KUKA KRL program: PPR_fullpath_2mm_split1.src

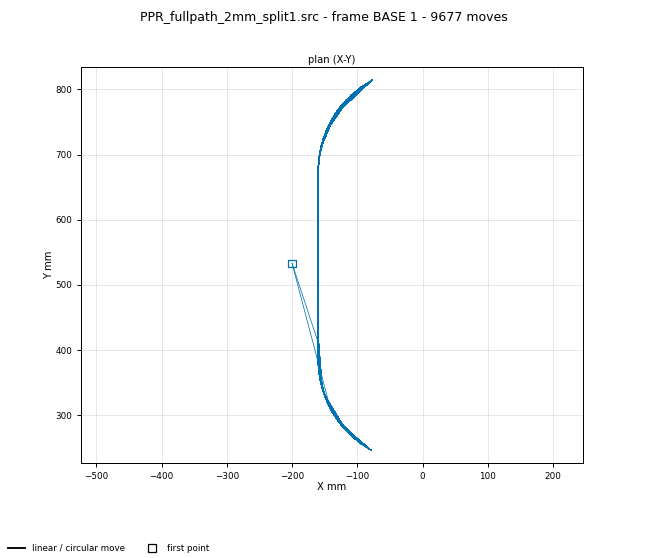
[picture p0: tool path of PPR_fullpath_2mm_split1.src in frame BASE 1, 9677 of 9678 moves have a stored position in this frame; points joined in program order, loops and branches not executed]
&ACCESS RVEO
&REL 11
&PARAM TEMPLATE = C:\KRC\Roboter\Template\vorgabe
&PARAM EDITMASK = *
DEF variable_helical2( )
;FOLD INI
  ;FOLD BASISTECH INI
    GLOBAL INTERRUPT DECL 3 WHEN $STOPMESS==TRUE DO IR_STOPM ( )
    INTERRUPT ON 3
    BAS (#INITMOV,0 )
  ;ENDFOLD (BASISTECH INI)
 ;FOLD USER INI


    ;Make your modifications here
  ;ENDFOLD (USER INI)
;ENDFOLD (INI)
ACTION(#AXIS_RESET,34,1000,#NOERROR,ERROR_CODE)
;FOLD PTP HOME  Vel= 100 % DEFAULT;%{PE}%MKUKATPBASIS,%CMOVE,%VPTP,%P 1:PTP, 2:HOME, 3:, 5:100, 7:DEFAULT
$BWDSTART = FALSE
PDAT_ACT=PDEFAULT
FDAT_ACT=FHOME
BAS (#PTP_PARAMS,100 )
$H_POS=XHOME
PTP  XHOME
;ENDFOLD
BAS(#TOOL,1)
BAS(#BASE,1)
$VEL_AXIS[1]=100
$VEL_AXIS[2]=100
$VEL_AXIS[3]=100
$VEL_AXIS[4]=100
$VEL_AXIS[5]=100
$VEL_AXIS[6]=100
$VEL_EXTAX[1]=100
$VEL_EXTAX[2]=100

$ACC_AXIS[1]=100
$ACC_AXIS[2]=100
$ACC_AXIS[3]=100
$ACC_AXIS[4]=100
$ACC_AXIS[5]=100
$ACC_AXIS[6]=100
$ACC_EXTAX[1]=100
$ACC_EXTAX[2]=100

SLIN {X  -200.000, Y  +533.000, Z    +0.000, A    +0.000, E1    +0.000, E3    +0.000, E4    +0.000}

SLIN {X  -141.408, Y  +310.842, Z    +0.000, E1   +71.243, E3  -388.598}
HALT
SPLINE
SPL {X  -134.330, Y  +298.778, Z    +0.000, E1   +70.323, E3  -374.632}
SPL {X  -128.957, Y  +290.989, Z    +0.000, E1   +69.528, E3  -365.267}
SPL {X  -124.846, Y  +285.632, Z    +0.000, E1   +68.906, E3  -358.804}
SPL {X  -121.783, Y  +281.927, Z    +0.000, E1   +68.403, E3  -354.372}
SPL {X   -79.219, Y  +246.688, Z    +0.000, E1   +55.887, E3  -232.865}
ENDSPLINE

SPLINE
SPL {X  -125.038, Y  +285.873, Z    +0.000, E1   +53.023, E3   -55.824}
SPL {X  -149.949, Y  +329.886, Z    +0.000, E1   +41.515, E3   -34.259}
SPL {X  -157.246, Y  +356.141, Z    +0.000, E1   +27.282, E3   -29.202}
SPL {X  -159.525, Y  +373.376, Z    +0.000, E1   +13.812, E3   -27.545}
SPL {X  -160.000, Y  +387.264, Z    +0.000, E1    +0.544, E3   -27.088}
SPL {X  -160.000, Y  +390.384, Z    +0.000, E1    -6.008, E3   -27.050}
SPL {X  -160.000, Y  +395.752, Z    +0.000, E1   -19.038, E3   -26.857}
SPL {X  -160.000, Y  +404.289, Z    +0.000, E1   -38.292, E3   -26.188}
SPL {X  -160.000, Y  +418.681, Z    +0.000, E1   -56.949, E3   -23.999}
SPL {X  -160.000, Y  +471.977, Z    +0.000, E1   -70.792, E3    -7.479}
SPL {X  -159.977, Y  +677.138, Z    +0.000, E1   -73.665, E3   +89.012}
SPL {X  -157.805, Y  +700.810, Z    +0.000, E1   -73.511, E3  +105.842}
SPL {X  -152.242, Y  +723.618, Z    +0.000, E1   -72.940, E3  +125.755}
SPL {X  -145.929, Y  +740.010, Z    +0.000, E1   -72.229, E3  +142.226}
SPL {X  -139.114, Y  +753.439, Z    +0.000, E1   -71.436, E3  +156.865}
SPL {X  -132.333, Y  +764.333, Z    +0.000, E1   -70.535, E3  +169.489}
SPL {X  -125.486, Y  +773.664, Z    +0.000, E1   -69.598, E3  +180.463}
SPL {X  -121.321, Y  +778.713, Z    +0.000, E1   -68.872, E3  +186.473}
SPL {X   -77.337, Y  +814.468, Z    +0.000, E1   -56.377, E3  +305.104}
ENDSPLINE

SPLINE
SPL {X  -134.727, Y  +760.706, Z    +0.000, E1   -50.460, E3  +493.336}
SPL {X  -155.580, Y  +711.748, Z    +0.000, E1   -32.084, E3  +510.251}
SPL {X  -159.445, Y  +687.715, Z    +0.000, E1   -14.660, E3  +513.097}
SPL {X  -159.995, Y  +675.725, Z    +0.000, E1    -3.424, E3  +513.608}
SPL {X  -160.000, Y  +671.714, Z    +0.000, E1    +0.835, E3  +513.649}
SPL {X  -160.000, Y  +663.084, Z    +0.000, E1   +21.134, E3  +513.973}
SPL {X  -160.000, Y  +650.910, Z    +0.000, E1   +46.005, E3  +515.127}
SPL {X  -160.000, Y  +634.843, Z    +0.000, E1   +61.273, E3  +517.804}
SPL {X  -160.000, Y  +578.679, Z    +0.000, E1   +71.665, E3  +535.637}
SPL {X  -160.000, Y  +387.528, Z    +0.000, E1   +73.487, E3  +628.450}
SPL {X  -159.218, Y  +369.903, Z    +0.000, E1   +73.425, E3  +640.317}
SPL {X  -156.808, Y  +353.900, Z    +0.000, E1   +73.180, E3  +652.921}
SPL {X  -154.539, Y  +344.254, Z    +0.000, E1   +72.827, E3  +662.458}
ENDSPLINE

SPLINE
SPL {X  -157.258, Y  +356.206, Z    +0.000, E1   +70.434, E3  +677.030}
ENDSPLINE

SPLINE
SPL {X  -150.342, Y  +330.952, Z    +0.000, E1   +71.154, E3  +688.703}
SPL {X  -141.358, Y  +310.748, Z    +0.000, E1   +71.233, E3  +701.409}
SPL {X  -134.330, Y  +298.778, Z    +0.000, E1   +70.323, E3  +715.256}
SPL {X  -128.957, Y  +290.989, Z    +0.000, E1   +69.528, E3  +724.621}
SPL {X  -124.846, Y  +285.632, Z    +0.000, E1   +68.906, E3  +731.084}
SPL {X  -121.783, Y  +281.927, Z    +0.000, E1   +68.403, E3  +735.517}
SPL {X   -79.219, Y  +246.688, Z    +0.000, E1   +55.887, E3  +857.023}
ENDSPLINE

SPLINE
SPL {X  -125.038, Y  +285.873, Z    +0.000, E1   +53.023, E3 +1034.064}
SPL {X  -149.949, Y  +329.886, Z    +0.000, E1   +41.515, E3 +1055.629}
SPL {X  -157.246, Y  +356.141, Z    +0.000, E1   +27.282, E3 +1060.686}
SPL {X  -159.525, Y  +373.376, Z    +0.000, E1   +13.812, E3 +1062.343}
SPL {X  -160.000, Y  +387.264, Z    +0.000, E1    +0.544, E3 +1062.800}
SPL {X  -160.000, Y  +390.384, Z    +0.000, E1    -6.008, E3 +1062.838}
SPL {X  -160.000, Y  +395.752, Z    +0.000, E1   -19.038, E3 +1063.031}
SPL {X  -160.000, Y  +404.289, Z    +0.000, E1   -38.292, E3 +1063.700}
SPL {X  -160.000, Y  +418.681, Z    +0.000, E1   -56.949, E3 +1065.889}
SPL {X  -160.000, Y  +471.977, Z    +0.000, E1   -70.792, E3 +1082.409}
SPL {X  -159.977, Y  +677.138, Z    +0.000, E1   -73.665, E3 +1178.900}
SPL {X  -157.805, Y  +700.810, Z    +0.000, E1   -73.511, E3 +1195.730}
SPL {X  -152.242, Y  +723.618, Z    +0.000, E1   -72.940, E3 +1215.643}
SPL {X  -145.929, Y  +740.010, Z    +0.000, E1   -72.229, E3 +1232.114}
SPL {X  -139.114, Y  +753.439, Z    +0.000, E1   -71.436, E3 +1246.753}
SPL {X  -132.333, Y  +764.333, Z    +0.000, E1   -70.535, E3 +1259.377}
SPL {X  -125.486, Y  +773.664, Z    +0.000, E1   -69.598, E3 +1270.351}
SPL {X  -121.321, Y  +778.713, Z    +0.000, E1   -68.872, E3 +1276.361}
SPL {X   -77.337, Y  +814.468, Z    +0.000, E1   -56.377, E3 +1394.992}
ENDSPLINE

SPLINE
SPL {X  -134.727, Y  +760.706, Z    +0.000, E1   -50.460, E3 +1583.224}
SPL {X  -155.580, Y  +711.748, Z    +0.000, E1   -32.084, E3 +1600.139}
SPL {X  -159.445, Y  +687.715, Z    +0.000, E1   -14.660, E3 +1602.986}
SPL {X  -159.995, Y  +675.725, Z    +0.000, E1    -3.424, E3 +1603.496}
SPL {X  -160.000, Y  +671.714, Z    +0.000, E1    +0.835, E3 +1603.537}
SPL {X  -160.000, Y  +663.084, Z    +0.000, E1   +21.134, E3 +1603.861}
SPL {X  -160.000, Y  +650.910, Z    +0.000, E1   +46.005, E3 +1605.015}
SPL {X  -160.000, Y  +634.843, Z    +0.000, E1   +61.273, E3 +1607.692}
SPL {X  -160.000, Y  +578.679, Z    +0.000, E1   +71.665, E3 +1625.525}
SPL {X  -160.000, Y  +387.528, Z    +0.000, E1   +73.487, E3 +1718.338}
SPL {X  -159.218, Y  +369.903, Z    +0.000, E1   +73.425, E3 +1730.205}
SPL {X  -156.808, Y  +353.900, Z    +0.000, E1   +73.180, E3 +1742.809}
SPL {X  -154.539, Y  +344.254, Z    +0.000, E1   +72.827, E3 +1752.346}
ENDSPLINE

SPLINE
SPL {X  -157.258, Y  +356.206, Z    +0.000, E1   +70.434, E3 +1766.919}
ENDSPLINE

SPLINE
SPL {X  -150.342, Y  +330.952, Z    +0.000, E1   +71.154, E3 +1778.591}
SPL {X  -141.358, Y  +310.748, Z    +0.000, E1   +71.233, E3 +1791.297}
SPL {X  -134.330, Y  +298.778, Z    +0.000, E1   +70.323, E3 +1805.144}
SPL {X  -128.957, Y  +290.989, Z    +0.000, E1   +69.528, E3 +1814.509}
SPL {X  -124.846, Y  +285.632, Z    +0.000, E1   +68.906, E3 +1820.972}
SPL {X  -121.783, Y  +281.927, Z    +0.000, E1   +68.403, E3 +1825.405}
SPL {X   -79.219, Y  +246.688, Z    +0.000, E1   +55.887, E3 +1946.911}
ENDSPLINE

SPLINE
SPL {X  -125.038, Y  +285.873, Z    +0.000, E1   +53.023, E3 +2123.952}
SPL {X  -149.949, Y  +329.886, Z    +0.000, E1   +41.515, E3 +2145.517}
SPL {X  -157.246, Y  +356.141, Z    +0.000, E1   +27.282, E3 +2150.574}
SPL {X  -159.525, Y  +373.376, Z    +0.000, E1   +13.812, E3 +2152.231}
SPL {X  -160.000, Y  +387.264, Z    +0.000, E1    +0.544, E3 +2152.688}
SPL {X  -160.000, Y  +390.384, Z    +0.000, E1    -6.008, E3 +2152.726}
SPL {X  -160.000, Y  +395.752, Z    +0.000, E1   -19.038, E3 +2152.919}
SPL {X  -160.000, Y  +404.289, Z    +0.000, E1   -38.292, E3 +2153.588}
SPL {X  -160.000, Y  +418.681, Z    +0.000, E1   -56.949, E3 +2155.777}
SPL {X  -160.000, Y  +471.977, Z    +0.000, E1   -70.792, E3 +2172.297}
SPL {X  -159.977, Y  +677.138, Z    +0.000, E1   -73.665, E3 +2268.788}
SPL {X  -157.805, Y  +700.810, Z    +0.000, E1   -73.511, E3 +2285.618}
SPL {X  -152.242, Y  +723.618, Z    +0.000, E1   -72.940, E3 +2305.531}
SPL {X  -145.929, Y  +740.010, Z    +0.000, E1   -72.229, E3 +2322.002}
SPL {X  -139.114, Y  +753.439, Z    +0.000, E1   -71.436, E3 +2336.641}
SPL {X  -132.333, Y  +764.333, Z    +0.000, E1   -70.535, E3 +2349.265}
SPL {X  -125.486, Y  +773.664, Z    +0.000, E1   -69.598, E3 +2360.239}
SPL {X  -121.321, Y  +778.713, Z    +0.000, E1   -68.872, E3 +2366.249}
SPL {X   -77.337, Y  +814.468, Z    +0.000, E1   -56.377, E3 +2484.880}
ENDSPLINE

SPLINE
SPL {X  -134.727, Y  +760.706, Z    +0.000, E1   -50.460, E3 +2673.112}
SPL {X  -155.580, Y  +711.748, Z    +0.000, E1   -32.084, E3 +2690.027}
SPL {X  -159.445, Y  +687.715, Z    +0.000, E1   -14.660, E3 +2692.874}
SPL {X  -159.995, Y  +675.725, Z    +0.000, E1    -3.424, E3 +2693.384}
SPL {X  -160.000, Y  +671.714, Z    +0.000, E1    +0.835, E3 +2693.425}
SPL {X  -160.000, Y  +663.084, Z    +0.000, E1   +21.134, E3 +2693.749}
SPL {X  -160.000, Y  +650.910, Z    +0.000, E1   +46.005, E3 +2694.903}
SPL {X  -160.000, Y  +634.843, Z    +0.000, E1   +61.273, E3 +2697.580}
SPL {X  -160.000, Y  +578.679, Z    +0.000, E1   +71.665, E3 +2715.413}
SPL {X  -160.000, Y  +387.528, Z    +0.000, E1   +73.487, E3 +2808.226}
SPL {X  -159.218, Y  +369.903, Z    +0.000, E1   +73.425, E3 +2820.093}
SPL {X  -156.808, Y  +353.900, Z    +0.000, E1   +73.180, E3 +2832.697}
SPL {X  -154.539, Y  +344.254, Z    +0.000, E1   +72.827, E3 +2842.234}
ENDSPLINE

SPLINE
SPL {X  -157.258, Y  +356.206, Z    +0.000, E1   +70.434, E3 +2856.807}
ENDSPLINE

SPLINE
SPL {X  -150.342, Y  +330.952, Z    +0.000, E1   +71.154, E3 +2868.479}
SPL {X  -141.358, Y  +310.748, Z    +0.000, E1   +71.233, E3 +2881.185}
SPL {X  -134.330, Y  +298.778, Z    +0.000, E1   +70.323, E3 +2895.032}
SPL {X  -128.957, Y  +290.989, Z    +0.000, E1   +69.528, E3 +2904.397}
SPL {X  -124.846, Y  +285.632, Z    +0.000, E1   +68.906, E3 +2910.860}
SPL {X  -121.783, Y  +281.927, Z    +0.000, E1   +68.403, E3 +2915.293}
SPL {X   -79.219, Y  +246.688, Z    +0.000, E1   +55.887, E3 +3036.799}
ENDSPLINE

SPLINE
SPL {X  -125.038, Y  +285.873, Z    +0.000, E1   +53.023, E3 +3213.840}
SPL {X  -149.949, Y  +329.886, Z    +0.000, E1   +41.515, E3 +3235.405}
SPL {X  -157.246, Y  +356.141, Z    +0.000, E1   +27.282, E3 +3240.462}
SPL {X  -159.525, Y  +373.376, Z    +0.000, E1   +13.812, E3 +3242.119}
SPL {X  -160.000, Y  +387.264, Z    +0.000, E1    +0.544, E3 +3242.577}
SPL {X  -160.000, Y  +390.384, Z    +0.000, E1    -6.008, E3 +3242.614}
SPL {X  -160.000, Y  +395.752, Z    +0.000, E1   -19.038, E3 +3242.807}
SPL {X  -160.000, Y  +404.289, Z    +0.000, E1   -38.292, E3 +3243.476}
SPL {X  -160.000, Y  +418.681, Z    +0.000, E1   -56.949, E3 +3245.665}
SPL {X  -160.000, Y  +458.961, Z    +0.000, E1   -69.778, E3 +3257.262}
SPL {X  -160.000, Y  +485.343, Z    +0.000, E1   -71.539, E3 +3267.248}
SPL {X  -159.977, Y  +677.138, Z    +0.000, E1   -73.665, E3 +3358.676}
SPL {X  -157.805, Y  +700.810, Z    +0.000, E1   -73.511, E3 +3375.506}
SPL {X  -152.242, Y  +723.618, Z    +0.000, E1   -72.940, E3 +3395.419}
SPL {X  -145.929, Y  +740.010, Z    +0.000, E1   -72.229, E3 +3411.890}
SPL {X  -139.114, Y  +753.439, Z    +0.000, E1   -71.436, E3 +3426.529}
SPL {X  -132.333, Y  +764.333, Z    +0.000, E1   -70.535, E3 +3439.153}
SPL {X  -125.486, Y  +773.664, Z    +0.000, E1   -69.598, E3 +3450.127}
SPL {X  -121.321, Y  +778.713, Z    +0.000, E1   -68.872, E3 +3456.137}
SPL {X   -77.337, Y  +814.468, Z    +0.000, E1   -56.377, E3 +3574.768}
ENDSPLINE

SPLINE
SPL {X  -134.727, Y  +760.706, Z    +0.000, E1   -50.460, E3 +3763.000}
SPL {X  -155.580, Y  +711.748, Z    +0.000, E1   -32.084, E3 +3779.915}
SPL {X  -159.445, Y  +687.715, Z    +0.000, E1   -14.660, E3 +3782.762}
SPL {X  -159.995, Y  +675.725, Z    +0.000, E1    -3.424, E3 +3783.272}
SPL {X  -160.000, Y  +671.714, Z    +0.000, E1    +0.835, E3 +3783.313}
SPL {X  -160.000, Y  +663.084, Z    +0.000, E1   +21.134, E3 +3783.637}
SPL {X  -160.000, Y  +650.910, Z    +0.000, E1   +46.005, E3 +3784.791}
SPL {X  -160.000, Y  +634.843, Z    +0.000, E1   +61.273, E3 +3787.468}
SPL {X  -160.000, Y  +578.679, Z    +0.000, E1   +71.665, E3 +3805.301}
SPL {X  -160.000, Y  +387.528, Z    +0.000, E1   +73.487, E3 +3898.114}
SPL {X  -159.218, Y  +369.903, Z    +0.000, E1   +73.425, E3 +3909.981}
SPL {X  -156.808, Y  +353.900, Z    +0.000, E1   +73.180, E3 +3922.585}
SPL {X  -154.539, Y  +344.254, Z    +0.000, E1   +72.827, E3 +3932.122}
ENDSPLINE

SPLINE
SPL {X  -157.258, Y  +356.206, Z    +0.000, E1   +70.434, E3 +3946.695}
ENDSPLINE

SPLINE
SPL {X  -150.342, Y  +330.952, Z    +0.000, E1   +71.154, E3 +3958.367}
SPL {X  -141.358, Y  +310.748, Z    +0.000, E1   +71.233, E3 +3971.073}
SPL {X  -134.330, Y  +298.778, Z    +0.000, E1   +70.323, E3 +3984.920}
SPL {X  -128.957, Y  +290.989, Z    +0.000, E1   +69.528, E3 +3994.285}
SPL {X  -124.846, Y  +285.632, Z    +0.000, E1   +68.906, E3 +4000.748}
SPL {X  -121.783, Y  +281.927, Z    +0.000, E1   +68.403, E3 +4005.181}
SPL {X   -79.219, Y  +246.688, Z    +0.000, E1   +55.887, E3 +4126.687}
ENDSPLINE

SPLINE
SPL {X  -125.038, Y  +285.873, Z    +0.000, E1   +53.023, E3 +4303.728}
SPL {X  -149.949, Y  +329.886, Z    +0.000, E1   +41.515, E3 +4325.293}
SPL {X  -157.246, Y  +356.141, Z    +0.000, E1   +27.282, E3 +4330.350}
SPL {X  -159.525, Y  +373.376, Z    +0.000, E1   +13.812, E3 +4332.007}
SPL {X  -160.000, Y  +387.264, Z    +0.000, E1    +0.544, E3 +4332.465}
SPL {X  -160.000, Y  +390.384, Z    +0.000, E1    -6.008, E3 +4332.502}
SPL {X  -160.000, Y  +395.752, Z    +0.000, E1   -19.038, E3 +4332.695}
SPL {X  -160.000, Y  +404.289, Z    +0.000, E1   -38.292, E3 +4333.364}
SPL {X  -160.000, Y  +418.681, Z    +0.000, E1   -56.949, E3 +4335.554}
SPL {X  -160.000, Y  +471.977, Z    +0.000, E1   -70.792, E3 +4352.073}
SPL {X  -159.977, Y  +677.138, Z    +0.000, E1   -73.665, E3 +4448.564}
SPL {X  -157.805, Y  +700.810, Z    +0.000, E1   -73.511, E3 +4465.394}
SPL {X  -152.242, Y  +723.618, Z    +0.000, E1   -72.940, E3 +4485.307}
SPL {X  -145.929, Y  +740.010, Z    +0.000, E1   -72.229, E3 +4501.778}
SPL {X  -139.114, Y  +753.439, Z    +0.000, E1   -71.436, E3 +4516.417}
SPL {X  -132.333, Y  +764.333, Z    +0.000, E1   -70.535, E3 +4529.041}
SPL {X  -125.486, Y  +773.664, Z    +0.000, E1   -69.598, E3 +4540.015}
SPL {X  -121.321, Y  +778.713, Z    +0.000, E1   -68.872, E3 +4546.025}
SPL {X   -77.337, Y  +814.468, Z    +0.000, E1   -56.377, E3 +4664.656}
ENDSPLINE

SPLINE
SPL {X  -134.727, Y  +760.706, Z    +0.000, E1   -50.460, E3 +4852.888}
SPL {X  -155.580, Y  +711.748, Z    +0.000, E1   -32.084, E3 +4869.803}
SPL {X  -159.445, Y  +687.715, Z    +0.000, E1   -14.660, E3 +4872.650}
SPL {X  -159.995, Y  +675.725, Z    +0.000, E1    -3.424, E3 +4873.160}
SPL {X  -160.000, Y  +671.714, Z    +0.000, E1    +0.835, E3 +4873.201}
SPL {X  -160.000, Y  +663.084, Z    +0.000, E1   +21.134, E3 +4873.525}
SPL {X  -160.000, Y  +650.910, Z    +0.000, E1   +46.005, E3 +4874.679}
SPL {X  -160.000, Y  +634.843, Z    +0.000, E1   +61.273, E3 +4877.356}
SPL {X  -160.000, Y  +578.679, Z    +0.000, E1   +71.665, E3 +4895.189}
SPL {X  -160.000, Y  +387.528, Z    +0.000, E1   +73.487, E3 +4988.002}
SPL {X  -159.218, Y  +369.903, Z    +0.000, E1   +73.425, E3 +4999.869}
SPL {X  -156.808, Y  +353.900, Z    +0.000, E1   +73.180, E3 +5012.473}
SPL {X  -154.539, Y  +344.254, Z    +0.000, E1   +72.827, E3 +5022.010}
ENDSPLINE

SPLINE
SPL {X  -157.258, Y  +356.206, Z    +0.000, E1   +70.434, E3 +5036.583}
ENDSPLINE

SPLINE
SPL {X  -150.342, Y  +330.952, Z    +0.000, E1   +71.154, E3 +5048.255}
SPL {X  -141.358, Y  +310.748, Z    +0.000, E1   +71.233, E3 +5060.961}
SPL {X  -134.330, Y  +298.778, Z    +0.000, E1   +70.323, E3 +5074.808}
SPL {X  -128.957, Y  +290.989, Z    +0.000, E1   +69.528, E3 +5084.173}
SPL {X  -124.846, Y  +285.632, Z    +0.000, E1   +68.906, E3 +5090.636}
SPL {X  -121.783, Y  +281.927, Z    +0.000, E1   +68.403, E3 +5095.069}
SPL {X   -79.219, Y  +246.688, Z    +0.000, E1   +55.887, E3 +5216.575}
ENDSPLINE

SPLINE
SPL {X  -125.038, Y  +285.873, Z    +0.000, E1   +53.023, E3 +5393.616}
SPL {X  -149.949, Y  +329.886, Z    +0.000, E1   +41.515, E3 +5415.181}
SPL {X  -157.246, Y  +356.141, Z    +0.000, E1   +27.282, E3 +5420.238}
SPL {X  -159.525, Y  +373.376, Z    +0.000, E1   +13.812, E3 +5421.895}
SPL {X  -160.000, Y  +387.264, Z    +0.000, E1    +0.544, E3 +5422.353}
SPL {X  -160.000, Y  +390.384, Z    +0.000, E1    -6.008, E3 +5422.390}
SPL {X  -160.000, Y  +395.752, Z    +0.000, E1   -19.038, E3 +5422.583}
SPL {X  -160.000, Y  +404.289, Z    +0.000, E1   -38.292, E3 +5423.252}
SPL {X  -160.000, Y  +418.681, Z    +0.000, E1   -56.949, E3 +5425.442}
SPL {X  -160.000, Y  +471.977, Z    +0.000, E1   -70.792, E3 +5441.961}
SPL {X  -159.977, Y  +677.138, Z    +0.000, E1   -73.665, E3 +5538.452}
SPL {X  -157.805, Y  +700.810, Z    +0.000, E1   -73.511, E3 +5555.282}
SPL {X  -152.242, Y  +723.618, Z    +0.000, E1   -72.940, E3 +5575.195}
SPL {X  -145.929, Y  +740.010, Z    +0.000, E1   -72.229, E3 +5591.666}
SPL {X  -139.114, Y  +753.439, Z    +0.000, E1   -71.436, E3 +5606.305}
SPL {X  -132.333, Y  +764.333, Z    +0.000, E1   -70.535, E3 +5618.929}
SPL {X  -125.486, Y  +773.664, Z    +0.000, E1   -69.598, E3 +5629.903}
SPL {X  -121.321, Y  +778.713, Z    +0.000, E1   -68.872, E3 +5635.913}
SPL {X   -77.337, Y  +814.468, Z    +0.000, E1   -56.377, E3 +5754.544}
ENDSPLINE

SPLINE
SPL {X  -134.727, Y  +760.706, Z    +0.000, E1   -50.460, E3 +5942.776}
SPL {X  -155.580, Y  +711.748, Z    +0.000, E1   -32.084, E3 +5959.691}
SPL {X  -159.445, Y  +687.715, Z    +0.000, E1   -14.660, E3 +5962.538}
SPL {X  -159.995, Y  +675.725, Z    +0.000, E1    -3.424, E3 +5963.048}
SPL {X  -160.000, Y  +671.714, Z    +0.000, E1    +0.835, E3 +5963.089}
SPL {X  -160.000, Y  +663.084, Z    +0.000, E1   +21.134, E3 +5963.413}
SPL {X  -160.000, Y  +650.910, Z    +0.000, E1   +46.005, E3 +5964.567}
SPL {X  -160.000, Y  +634.843, Z    +0.000, E1   +61.273, E3 +5967.244}
SPL {X  -160.000, Y  +578.679, Z    +0.000, E1   +71.665, E3 +5985.078}
SPL {X  -160.000, Y  +387.528, Z    +0.000, E1   +73.487, E3 +6077.890}
SPL {X  -159.218, Y  +369.903, Z    +0.000, E1   +73.425, E3 +6089.757}
SPL {X  -156.808, Y  +353.900, Z    +0.000, E1   +73.180, E3 +6102.361}
SPL {X  -154.539, Y  +344.254, Z    +0.000, E1   +72.827, E3 +6111.898}
ENDSPLINE

SPLINE
SPL {X  -157.258, Y  +356.206, Z    +0.000, E1   +70.434, E3 +6126.471}
ENDSPLINE

SPLINE
SPL {X  -150.342, Y  +330.952, Z    +0.000, E1   +71.154, E3 +6138.143}
SPL {X  -141.358, Y  +310.748, Z    +0.000, E1   +71.233, E3 +6150.849}
SPL {X  -134.330, Y  +298.778, Z    +0.000, E1   +70.323, E3 +6164.696}
SPL {X  -128.957, Y  +290.989, Z    +0.000, E1   +69.528, E3 +6174.061}
SPL {X  -124.846, Y  +285.632, Z    +0.000, E1   +68.906, E3 +6180.524}
SPL {X  -121.783, Y  +281.927, Z    +0.000, E1   +68.403, E3 +6184.957}
SPL {X   -79.219, Y  +246.688, Z    +0.000, E1   +55.887, E3 +6306.463}
ENDSPLINE

SPLINE
SPL {X  -125.038, Y  +285.873, Z    +0.000, E1   +53.023, E3 +6483.504}
SPL {X  -149.949, Y  +329.886, Z    +0.000, E1   +41.515, E3 +6505.069}
SPL {X  -157.246, Y  +356.141, Z    +0.000, E1   +27.282, E3 +6510.126}
SPL {X  -159.525, Y  +373.376, Z    +0.000, E1   +13.812, E3 +6511.783}
SPL {X  -160.000, Y  +387.264, Z    +0.000, E1    +0.544, E3 +6512.241}
SPL {X  -160.000, Y  +390.384, Z    +0.000, E1    -6.008, E3 +6512.278}
SPL {X  -160.000, Y  +395.752, Z    +0.000, E1   -19.038, E3 +6512.471}
SPL {X  -160.000, Y  +404.289, Z    +0.000, E1   -38.292, E3 +6513.140}
SPL {X  -160.000, Y  +418.681, Z    +0.000, E1   -56.949, E3 +6515.330}
SPL {X  -160.000, Y  +458.961, Z    +0.000, E1   -69.778, E3 +6526.926}
SPL {X  -160.000, Y  +485.343, Z    +0.000, E1   -71.539, E3 +6536.912}
SPL {X  -159.977, Y  +677.138, Z    +0.000, E1   -73.665, E3 +6628.340}
SPL {X  -157.805, Y  +700.810, Z    +0.000, E1   -73.511, E3 +6645.170}
SPL {X  -152.242, Y  +723.618, Z    +0.000, E1   -72.940, E3 +6665.083}
SPL {X  -145.929, Y  +740.010, Z    +0.000, E1   -72.229, E3 +6681.554}
SPL {X  -139.114, Y  +753.439, Z    +0.000, E1   -71.436, E3 +6696.193}
SPL {X  -132.333, Y  +764.333, Z    +0.000, E1   -70.535, E3 +6708.817}
SPL {X  -125.486, Y  +773.664, Z    +0.000, E1   -69.598, E3 +6719.791}
SPL {X  -121.321, Y  +778.713, Z    +0.000, E1   -68.872, E3 +6725.801}
SPL {X   -77.337, Y  +814.468, Z    +0.000, E1   -56.377, E3 +6844.432}
ENDSPLINE

SPLINE
SPL {X  -134.727, Y  +760.706, Z    +0.000, E1   -50.460, E3 +7032.664}
SPL {X  -155.580, Y  +711.748, Z    +0.000, E1   -32.084, E3 +7049.579}
SPL {X  -159.445, Y  +687.715, Z    +0.000, E1   -14.660, E3 +7052.426}
SPL {X  -159.995, Y  +675.725, Z    +0.000, E1    -3.424, E3 +7052.937}
SPL {X  -160.000, Y  +671.714, Z    +0.000, E1    +0.835, E3 +7052.977}
SPL {X  -160.000, Y  +663.084, Z    +0.000, E1   +21.134, E3 +7053.301}
SPL {X  -160.000, Y  +650.910, Z    +0.000, E1   +46.005, E3 +7054.455}
SPL {X  -160.000, Y  +634.843, Z    +0.000, E1   +61.273, E3 +7057.132}
SPL {X  -160.000, Y  +578.679, Z    +0.000, E1   +71.665, E3 +7074.966}
SPL {X  -160.000, Y  +387.528, Z    +0.000, E1   +73.487, E3 +7167.778}
SPL {X  -159.218, Y  +369.903, Z    +0.000, E1   +73.425, E3 +7179.645}
SPL {X  -156.808, Y  +353.900, Z    +0.000, E1   +73.180, E3 +7192.249}
SPL {X  -154.539, Y  +344.254, Z    +0.000, E1   +72.827, E3 +7201.786}
ENDSPLINE

SPLINE
SPL {X  -157.258, Y  +356.206, Z    +0.000, E1   +70.434, E3 +7216.359}
ENDSPLINE

SPLINE
SPL {X  -150.342, Y  +330.952, Z    +0.000, E1   +71.154, E3 +7228.031}
SPL {X  -141.358, Y  +310.748, Z    +0.000, E1   +71.233, E3 +7240.737}
SPL {X  -134.330, Y  +298.778, Z    +0.000, E1   +70.323, E3 +7254.584}
SPL {X  -128.957, Y  +290.989, Z    +0.000, E1   +69.528, E3 +7263.949}
SPL {X  -124.846, Y  +285.632, Z    +0.000, E1   +68.906, E3 +7270.413}
SPL {X  -121.783, Y  +281.927, Z    +0.000, E1   +68.403, E3 +7274.845}
SPL {X   -79.219, Y  +246.688, Z    +0.000, E1   +55.887, E3 +7396.351}
ENDSPLINE

SPLINE
SPL {X  -125.038, Y  +285.873, Z    +0.000, E1   +53.023, E3 +7573.392}
SPL {X  -149.949, Y  +329.886, Z    +0.000, E1   +41.515, E3 +7594.957}
SPL {X  -157.246, Y  +356.141, Z    +0.000, E1   +27.282, E3 +7600.014}
SPL {X  -159.525, Y  +373.376, Z    +0.000, E1   +13.812, E3 +7601.671}
SPL {X  -160.000, Y  +387.264, Z    +0.000, E1    +0.544, E3 +7602.129}
SPL {X  -160.000, Y  +390.384, Z    +0.000, E1    -6.008, E3 +7602.166}
SPL {X  -160.000, Y  +395.752, Z    +0.000, E1   -19.038, E3 +7602.359}
SPL {X  -160.000, Y  +404.289, Z    +0.000, E1   -38.292, E3 +7603.028}
SPL {X  -160.000, Y  +418.681, Z    +0.000, E1   -56.949, E3 +7605.218}
SPL {X  -160.000, Y  +471.977, Z    +0.000, E1   -70.792, E3 +7621.737}
SPL {X  -159.977, Y  +677.138, Z    +0.000, E1   -73.665, E3 +7718.228}
SPL {X  -157.805, Y  +700.810, Z    +0.000, E1   -73.511, E3 +7735.058}
SPL {X  -152.242, Y  +723.618, Z    +0.000, E1   -72.940, E3 +7754.971}
SPL {X  -145.929, Y  +740.010, Z    +0.000, E1   -72.229, E3 +7771.442}
SPL {X  -139.114, Y  +753.439, Z    +0.000, E1   -71.436, E3 +7786.081}
SPL {X  -132.333, Y  +764.333, Z    +0.000, E1   -70.535, E3 +7798.705}
SPL {X  -125.486, Y  +773.664, Z    +0.000, E1   -69.598, E3 +7809.679}
SPL {X  -121.321, Y  +778.713, Z    +0.000, E1   -68.872, E3 +7815.689}
SPL {X   -77.337, Y  +814.468, Z    +0.000, E1   -56.377, E3 +7934.320}
ENDSPLINE

SPLINE
SPL {X  -134.727, Y  +760.706, Z    +0.000, E1   -50.460, E3 +8122.552}
SPL {X  -155.580, Y  +711.748, Z    +0.000, E1   -32.084, E3 +8139.467}
SPL {X  -159.445, Y  +687.715, Z    +0.000, E1   -14.660, E3 +8142.314}
SPL {X  -159.995, Y  +675.725, Z    +0.000, E1    -3.424, E3 +8142.825}
SPL {X  -160.000, Y  +671.714, Z    +0.000, E1    +0.835, E3 +8142.865}
SPL {X  -160.000, Y  +663.084, Z    +0.000, E1   +21.134, E3 +8143.189}
SPL {X  -160.000, Y  +650.910, Z    +0.000, E1   +46.005, E3 +8144.343}
SPL {X  -160.000, Y  +634.843, Z    +0.000, E1   +61.273, E3 +8147.020}
SPL {X  -160.000, Y  +578.679, Z    +0.000, E1   +71.665, E3 +8164.854}
SPL {X  -160.000, Y  +387.528, Z    +0.000, E1   +73.487, E3 +8257.666}
SPL {X  -159.218, Y  +369.903, Z    +0.000, E1   +73.425, E3 +8269.533}
SPL {X  -156.808, Y  +353.900, Z    +0.000, E1   +73.180, E3 +8282.137}
SPL {X  -154.539, Y  +344.254, Z    +0.000, E1   +72.827, E3 +8291.674}
ENDSPLINE

SPLINE
SPL {X  -157.258, Y  +356.206, Z    +0.000, E1   +70.434, E3 +8306.247}
ENDSPLINE

SPLINE
SPL {X  -150.342, Y  +330.952, Z    +0.000, E1   +71.154, E3 +8317.919}
SPL {X  -141.358, Y  +310.748, Z    +0.000, E1   +71.233, E3 +8330.625}
SPL {X  -134.330, Y  +298.778, Z    +0.000, E1   +70.323, E3 +8344.472}
SPL {X  -128.957, Y  +290.989, Z    +0.000, E1   +69.528, E3 +8353.837}
SPL {X  -124.846, Y  +285.632, Z    +0.000, E1   +68.906, E3 +8360.301}
SPL {X  -121.783, Y  +281.927, Z    +0.000, E1   +68.403, E3 +8364.733}
SPL {X   -79.219, Y  +246.688, Z    +0.000, E1   +55.887, E3 +8486.239}
ENDSPLINE

SPLINE
SPL {X  -125.038, Y  +285.873, Z    +0.000, E1   +53.023, E3 +8663.280}
SPL {X  -149.949, Y  +329.886, Z    +0.000, E1   +41.515, E3 +8684.845}
SPL {X  -157.246, Y  +356.141, Z    +0.000, E1   +27.282, E3 +8689.902}
SPL {X  -159.525, Y  +373.376, Z    +0.000, E1   +13.812, E3 +8691.559}
SPL {X  -160.000, Y  +387.264, Z    +0.000, E1    +0.544, E3 +8692.017}
SPL {X  -160.000, Y  +390.384, Z    +0.000, E1    -6.008, E3 +8692.054}
SPL {X  -160.000, Y  +395.752, Z    +0.000, E1   -19.038, E3 +8692.248}
SPL {X  -160.000, Y  +404.289, Z    +0.000, E1   -38.292, E3 +8692.916}
SPL {X  -160.000, Y  +418.681, Z    +0.000, E1   -56.949, E3 +8695.106}
SPL {X  -160.000, Y  +471.977, Z    +0.000, E1   -70.792, E3 +8711.625}
SPL {X  -159.977, Y  +677.138, Z    +0.000, E1   -73.665, E3 +8808.116}
SPL {X  -157.805, Y  +700.810, Z    +0.000, E1   -73.511, E3 +8824.946}
SPL {X  -152.242, Y  +723.618, Z    +0.000, E1   -72.940, E3 +8844.859}
SPL {X  -145.929, Y  +740.010, Z    +0.000, E1   -72.229, E3 +8861.331}
SPL {X  -139.114, Y  +753.439, Z    +0.000, E1   -71.436, E3 +8875.969}
SPL {X  -132.333, Y  +764.333, Z    +0.000, E1   -70.535, E3 +8888.593}
SPL {X  -125.486, Y  +773.664, Z    +0.000, E1   -69.598, E3 +8899.567}
SPL {X  -121.321, Y  +778.713, Z    +0.000, E1   -68.872, E3 +8905.577}
SPL {X   -77.337, Y  +814.468, Z    +0.000, E1   -56.377, E3 +9024.208}
ENDSPLINE

SPLINE
SPL {X  -134.727, Y  +760.706, Z    +0.000, E1   -50.460, E3 +9212.440}
SPL {X  -155.580, Y  +711.748, Z    +0.000, E1   -32.084, E3 +9229.355}
SPL {X  -159.445, Y  +687.715, Z    +0.000, E1   -14.660, E3 +9232.202}
SPL {X  -159.995, Y  +675.725, Z    +0.000, E1    -3.424, E3 +9232.713}
SPL {X  -160.000, Y  +671.714, Z    +0.000, E1    +0.835, E3 +9232.753}
SPL {X  -160.000, Y  +663.084, Z    +0.000, E1   +21.134, E3 +9233.077}
SPL {X  -160.000, Y  +650.910, Z    +0.000, E1   +46.005, E3 +9234.231}
SPL {X  -160.000, Y  +634.843, Z    +0.000, E1   +61.273, E3 +9236.908}
SPL {X  -160.000, Y  +578.679, Z    +0.000, E1   +71.665, E3 +9254.742}
SPL {X  -160.000, Y  +387.528, Z    +0.000, E1   +73.487, E3 +9347.554}
SPL {X  -159.218, Y  +369.903, Z    +0.000, E1   +73.425, E3 +9359.421}
SPL {X  -156.808, Y  +353.900, Z    +0.000, E1   +73.180, E3 +9372.025}
SPL {X  -154.539, Y  +344.254, Z    +0.000, E1   +72.827, E3 +9381.562}
ENDSPLINE

SPLINE
SPL {X  -157.258, Y  +356.206, Z    +0.000, E1   +70.434, E3 +9396.135}
ENDSPLINE

SPLINE
SPL {X  -150.342, Y  +330.952, Z    +0.000, E1   +71.154, E3 +9407.807}
SPL {X  -141.358, Y  +310.748, Z    +0.000, E1   +71.233, E3 +9420.513}
SPL {X  -134.330, Y  +298.778, Z    +0.000, E1   +70.323, E3 +9434.360}
SPL {X  -128.957, Y  +290.989, Z    +0.000, E1   +69.528, E3 +9443.725}
SPL {X  -124.846, Y  +285.632, Z    +0.000, E1   +68.906, E3 +9450.189}
SPL {X  -121.783, Y  +281.927, Z    +0.000, E1   +68.403, E3 +9454.621}
SPL {X   -79.219, Y  +246.688, Z    +0.000, E1   +55.887, E3 +9576.127}
ENDSPLINE

SPLINE
SPL {X  -125.038, Y  +285.873, Z    +0.000, E1   +53.023, E3 +9753.168}
SPL {X  -149.949, Y  +329.886, Z    +0.000, E1   +41.515, E3 +9774.733}
SPL {X  -157.246, Y  +356.141, Z    +0.000, E1   +27.282, E3 +9779.790}
SPL {X  -159.525, Y  +373.376, Z    +0.000, E1   +13.812, E3 +9781.447}
SPL {X  -160.000, Y  +387.264, Z    +0.000, E1    +0.544, E3 +9781.905}
SPL {X  -160.000, Y  +390.384, Z    +0.000, E1    -6.008, E3 +9781.942}
SPL {X  -160.000, Y  +395.752, Z    +0.000, E1   -19.038, E3 +9782.136}
SPL {X  -160.000, Y  +404.289, Z    +0.000, E1   -38.292, E3 +9782.804}
SPL {X  -160.000, Y  +418.681, Z    +0.000, E1   -56.949, E3 +9784.994}
SPL {X  -160.000, Y  +471.977, Z    +0.000, E1   -70.792, E3 +9801.513}
SPL {X  -159.977, Y  +677.138, Z    +0.000, E1   -73.665, E3 +9898.004}
SPL {X  -157.805, Y  +700.810, Z    +0.000, E1   -73.511, E3 +9914.834}
SPL {X  -152.242, Y  +723.618, Z    +0.000, E1   -72.940, E3 +9934.747}
SPL {X  -145.929, Y  +740.010, Z    +0.000, E1   -72.229, E3 +9951.219}
SPL {X  -139.114, Y  +753.439, Z    +0.000, E1   -71.436, E3 +9965.857}
SPL {X  -132.333, Y  +764.333, Z    +0.000, E1   -70.535, E3 +9978.481}
SPL {X  -125.486, Y  +773.664, Z    +0.000, E1   -69.598, E3 +9989.455}
SPL {X  -121.321, Y  +778.713, Z    +0.000, E1   -68.872, E3 +9995.465}
SPL {X   -77.337, Y  +814.468, Z    +0.000, E1   -56.377, E3 +10114.097}
ENDSPLINE

SPLINE
SPL {X  -134.727, Y  +760.706, Z    +0.000, E1   -50.460, E3 +10302.328}
SPL {X  -155.580, Y  +711.748, Z    +0.000, E1   -32.084, E3 +10319.243}
SPL {X  -159.445, Y  +687.715, Z    +0.000, E1   -14.660, E3 +10322.090}
SPL {X  -159.995, Y  +675.725, Z    +0.000, E1    -3.424, E3 +10322.601}
SPL {X  -160.000, Y  +671.714, Z    +0.000, E1    +0.835, E3 +10322.641}
SPL {X  -160.000, Y  +663.084, Z    +0.000, E1   +21.134, E3 +10322.965}
SPL {X  -160.000, Y  +650.910, Z    +0.000, E1   +46.005, E3 +10324.119}
SPL {X  -160.000, Y  +634.843, Z    +0.000, E1   +61.273, E3 +10326.796}
SPL {X  -160.000, Y  +578.679, Z    +0.000, E1   +71.665, E3 +10344.630}
SPL {X  -160.000, Y  +387.528, Z    +0.000, E1   +73.487, E3 +10437.442}
SPL {X  -159.218, Y  +369.903, Z    +0.000, E1   +73.425, E3 +10449.309}
SPL {X  -156.808, Y  +353.900, Z    +0.000, E1   +73.180, E3 +10461.913}
SPL {X  -154.539, Y  +344.254, Z    +0.000, E1   +72.827, E3 +10471.450}
ENDSPLINE

SPLINE
SPL {X  -157.258, Y  +356.206, Z    +0.000, E1   +70.434, E3 +10486.023}
ENDSPLINE

SPLINE
SPL {X  -150.342, Y  +330.952, Z    +0.000, E1   +71.154, E3 +10497.695}
SPL {X  -141.358, Y  +310.748, Z    +0.000, E1   +71.233, E3 +10510.401}
SPL {X  -134.330, Y  +298.778, Z    +0.000, E1   +70.323, E3 +10524.248}
SPL {X  -128.957, Y  +290.989, Z    +0.000, E1   +69.528, E3 +10533.613}
SPL {X  -124.846, Y  +285.632, Z    +0.000, E1   +68.906, E3 +10540.077}
SPL {X  -121.783, Y  +281.927, Z    +0.000, E1   +68.403, E3 +10544.509}
SPL {X   -79.219, Y  +246.688, Z    +0.000, E1   +55.887, E3 +10666.015}
ENDSPLINE

SPLINE
SPL {X  -125.038, Y  +285.873, Z    +0.000, E1   +53.023, E3 +10843.056}
SPL {X  -149.949, Y  +329.886, Z    +0.000, E1   +41.515, E3 +10864.621}
SPL {X  -157.246, Y  +356.141, Z    +0.000, E1   +27.282, E3 +10869.678}
SPL {X  -159.525, Y  +373.376, Z    +0.000, E1   +13.812, E3 +10871.335}
SPL {X  -160.000, Y  +387.264, Z    +0.000, E1    +0.544, E3 +10871.793}
SPL {X  -160.000, Y  +390.384, Z    +0.000, E1    -6.008, E3 +10871.830}
SPL {X  -160.000, Y  +395.752, Z    +0.000, E1   -19.038, E3 +10872.024}
SPL {X  -160.000, Y  +404.289, Z    +0.000, E1   -38.292, E3 +10872.692}
SPL {X  -160.000, Y  +418.681, Z    +0.000, E1   -56.949, E3 +10874.882}
SPL {X  -160.000, Y  +471.977, Z    +0.000, E1   -70.792, E3 +10891.401}
SPL {X  -159.977, Y  +677.138, Z    +0.000, E1   -73.665, E3 +10987.892}
SPL {X  -157.805, Y  +700.810, Z    +0.000, E1   -73.511, E3 +11004.722}
SPL {X  -152.242, Y  +723.618, Z    +0.000, E1   -72.940, E3 +11024.635}
SPL {X  -145.929, Y  +740.010, Z    +0.000, E1   -72.229, E3 +11041.107}
SPL {X  -139.114, Y  +753.439, Z    +0.000, E1   -71.436, E3 +11055.745}
SPL {X  -132.333, Y  +764.333, Z    +0.000, E1   -70.535, E3 +11068.369}
SPL {X  -125.486, Y  +773.664, Z    +0.000, E1   -69.598, E3 +11079.343}
SPL {X  -121.321, Y  +778.713, Z    +0.000, E1   -68.872, E3 +11085.353}
SPL {X   -77.337, Y  +814.468, Z    +0.000, E1   -56.377, E3 +11203.985}
ENDSPLINE

SPLINE
SPL {X  -134.727, Y  +760.706, Z    +0.000, E1   -50.460, E3 +11392.216}
SPL {X  -155.580, Y  +711.748, Z    +0.000, E1   -32.084, E3 +11409.131}
SPL {X  -159.445, Y  +687.715, Z    +0.000, E1   -14.660, E3 +11411.978}
SPL {X  -159.995, Y  +675.725, Z    +0.000, E1    -3.424, E3 +11412.489}
SPL {X  -160.000, Y  +671.714, Z    +0.000, E1    +0.835, E3 +11412.529}
SPL {X  -160.000, Y  +663.084, Z    +0.000, E1   +21.134, E3 +11412.853}
SPL {X  -160.000, Y  +650.910, Z    +0.000, E1   +46.005, E3 +11414.007}
SPL {X  -160.000, Y  +634.843, Z    +0.000, E1   +61.273, E3 +11416.684}
SPL {X  -160.000, Y  +578.679, Z    +0.000, E1   +71.665, E3 +11434.518}
SPL {X  -160.000, Y  +387.528, Z    +0.000, E1   +73.487, E3 +11527.330}
SPL {X  -159.218, Y  +369.903, Z    +0.000, E1   +73.425, E3 +11539.197}
SPL {X  -156.808, Y  +353.900, Z    +0.000, E1   +73.180, E3 +11551.801}
SPL {X  -154.539, Y  +344.254, Z    +0.000, E1   +72.827, E3 +11561.338}
ENDSPLINE

SPLINE
SPL {X  -157.258, Y  +356.206, Z    +0.000, E1   +70.434, E3 +11575.911}
ENDSPLINE

SPLINE
SPL {X  -150.342, Y  +330.952, Z    +0.000, E1   +71.154, E3 +11587.583}
SPL {X  -141.358, Y  +310.748, Z    +0.000, E1   +71.233, E3 +11600.289}
SPL {X  -134.330, Y  +298.778, Z    +0.000, E1   +70.323, E3 +11614.136}
SPL {X  -128.957, Y  +290.989, Z    +0.000, E1   +69.528, E3 +11623.501}
SPL {X  -124.846, Y  +285.632, Z    +0.000, E1   +68.906, E3 +11629.965}
SPL {X  -121.783, Y  +281.927, Z    +0.000, E1   +68.403, E3 +11634.397}
SPL {X   -79.219, Y  +246.688, Z    +0.000, E1   +55.887, E3 +11755.903}
ENDSPLINE

SPLINE
SPL {X  -125.038, Y  +285.873, Z    +0.000, E1   +53.023, E3 +11932.944}
SPL {X  -149.949, Y  +329.886, Z    +0.000, E1   +41.515, E3 +11954.509}
SPL {X  -157.246, Y  +356.141, Z    +0.000, E1   +27.282, E3 +11959.566}
SPL {X  -159.525, Y  +373.376, Z    +0.000, E1   +13.812, E3 +11961.223}
SPL {X  -160.000, Y  +387.264, Z    +0.000, E1    +0.544, E3 +11961.681}
SPL {X  -160.000, Y  +390.384, Z    +0.000, E1    -6.008, E3 +11961.718}
SPL {X  -160.000, Y  +395.752, Z    +0.000, E1   -19.038, E3 +11961.912}
SPL {X  -160.000, Y  +404.289, Z    +0.000, E1   -38.292, E3 +11962.580}
SPL {X  -160.000, Y  +418.681, Z    +0.000, E1   -56.949, E3 +11964.770}
SPL {X  -160.000, Y  +471.977, Z    +0.000, E1   -70.792, E3 +11981.289}
SPL {X  -159.977, Y  +677.138, Z    +0.000, E1   -73.665, E3 +12077.780}
SPL {X  -157.805, Y  +700.810, Z    +0.000, E1   -73.511, E3 +12094.610}
SPL {X  -152.242, Y  +723.618, Z    +0.000, E1   -72.940, E3 +12114.523}
SPL {X  -145.929, Y  +740.010, Z    +0.000, E1   -72.229, E3 +12130.995}
SPL {X  -139.114, Y  +753.439, Z    +0.000, E1   -71.436, E3 +12145.633}
SPL {X  -132.333, Y  +764.333, Z    +0.000, E1   -70.535, E3 +12158.257}
SPL {X  -125.486, Y  +773.664, Z    +0.000, E1   -69.598, E3 +12169.231}
SPL {X  -121.321, Y  +778.713, Z    +0.000, E1   -68.872, E3 +12175.241}
SPL {X   -77.337, Y  +814.468, Z    +0.000, E1   -56.377, E3 +12293.873}
ENDSPLINE

SPLINE
SPL {X  -134.727, Y  +760.706, Z    +0.000, E1   -50.460, E3 +12482.104}
SPL {X  -155.580, Y  +711.748, Z    +0.000, E1   -32.084, E3 +12499.019}
SPL {X  -159.445, Y  +687.715, Z    +0.000, E1   -14.660, E3 +12501.866}
SPL {X  -159.995, Y  +675.725, Z    +0.000, E1    -3.424, E3 +12502.377}
SPL {X  -160.000, Y  +671.714, Z    +0.000, E1    +0.835, E3 +12502.417}
SPL {X  -160.000, Y  +663.084, Z    +0.000, E1   +21.134, E3 +12502.741}
SPL {X  -160.000, Y  +650.910, Z    +0.000, E1   +46.005, E3 +12503.895}
SPL {X  -160.000, Y  +634.843, Z    +0.000, E1   +61.273, E3 +12506.572}
SPL {X  -160.000, Y  +578.679, Z    +0.000, E1   +71.665, E3 +12524.406}
SPL {X  -160.000, Y  +387.528, Z    +0.000, E1   +73.487, E3 +12617.218}
SPL {X  -159.218, Y  +369.903, Z    +0.000, E1   +73.425, E3 +12629.085}
SPL {X  -156.808, Y  +353.900, Z    +0.000, E1   +73.180, E3 +12641.689}
SPL {X  -154.539, Y  +344.254, Z    +0.000, E1   +72.827, E3 +12651.226}
ENDSPLINE

SPLINE
SPL {X  -157.258, Y  +356.206, Z    +0.000, E1   +70.434, E3 +12665.799}
ENDSPLINE

SPLINE
SPL {X  -150.342, Y  +330.952, Z    +0.000, E1   +71.154, E3 +12677.471}
SPL {X  -141.358, Y  +310.748, Z    +0.000, E1   +71.233, E3 +12690.177}
SPL {X  -134.330, Y  +298.778, Z    +0.000, E1   +70.323, E3 +12704.024}
SPL {X  -128.957, Y  +290.989, Z    +0.000, E1   +69.528, E3 +12713.389}
SPL {X  -124.846, Y  +285.632, Z    +0.000, E1   +68.906, E3 +12719.853}
SPL {X  -121.783, Y  +281.927, Z    +0.000, E1   +68.403, E3 +12724.285}
SPL {X   -79.219, Y  +246.688, Z    +0.000, E1   +55.887, E3 +12845.791}
ENDSPLINE

SPLINE
SPL {X  -125.038, Y  +285.873, Z    +0.000, E1   +53.023, E3 +13022.832}
SPL {X  -149.949, Y  +329.886, Z    +0.000, E1   +41.515, E3 +13044.397}
SPL {X  -157.246, Y  +356.141, Z    +0.000, E1   +27.282, E3 +13049.454}
SPL {X  -159.525, Y  +373.376, Z    +0.000, E1   +13.812, E3 +13051.111}
SPL {X  -160.000, Y  +387.264, Z    +0.000, E1    +0.544, E3 +13051.569}
SPL {X  -160.000, Y  +390.384, Z    +0.000, E1    -6.008, E3 +13051.606}
SPL {X  -160.000, Y  +395.752, Z    +0.000, E1   -19.038, E3 +13051.800}
SPL {X  -160.000, Y  +404.289, Z    +0.000, E1   -38.292, E3 +13052.468}
SPL {X  -160.000, Y  +418.681, Z    +0.000, E1   -56.949, E3 +13054.658}
SPL {X  -160.000, Y  +471.977, Z    +0.000, E1   -70.792, E3 +13071.177}
SPL {X  -159.977, Y  +677.138, Z    +0.000, E1   -73.665, E3 +13167.668}
SPL {X  -157.805, Y  +700.810, Z    +0.000, E1   -73.511, E3 +13184.499}
SPL {X  -152.242, Y  +723.618, Z    +0.000, E1   -72.940, E3 +13204.411}
SPL {X  -145.929, Y  +740.010, Z    +0.000, E1   -72.229, E3 +13220.883}
SPL {X  -139.114, Y  +753.439, Z    +0.000, E1   -71.436, E3 +13235.521}
SPL {X  -132.333, Y  +764.333, Z    +0.000, E1   -70.535, E3 +13248.145}
SPL {X  -125.486, Y  +773.664, Z    +0.000, E1   -69.598, E3 +13259.119}
SPL {X  -121.321, Y  +778.713, Z    +0.000, E1   -68.872, E3 +13265.129}
SPL {X   -77.337, Y  +814.468, Z    +0.000, E1   -56.377, E3 +13383.761}
ENDSPLINE

SPLINE
SPL {X  -134.727, Y  +760.706, Z    +0.000, E1   -50.460, E3 +13571.993}
SPL {X  -155.580, Y  +711.748, Z    +0.000, E1   -32.084, E3 +13588.907}
SPL {X  -159.445, Y  +687.715, Z    +0.000, E1   -14.660, E3 +13591.754}
SPL {X  -159.995, Y  +675.725, Z    +0.000, E1    -3.424, E3 +13592.265}
SPL {X  -160.000, Y  +671.714, Z    +0.000, E1    +0.835, E3 +13592.305}
SPL {X  -160.000, Y  +663.084, Z    +0.000, E1   +21.134, E3 +13592.630}
SPL {X  -160.000, Y  +650.910, Z    +0.000, E1   +46.005, E3 +13593.783}
SPL {X  -160.000, Y  +634.843, Z    +0.000, E1   +61.273, E3 +13596.460}
SPL {X  -160.000, Y  +578.679, Z    +0.000, E1   +71.665, E3 +13614.294}
SPL {X  -160.000, Y  +387.528, Z    +0.000, E1   +73.487, E3 +13707.106}
SPL {X  -159.218, Y  +369.903, Z    +0.000, E1   +73.425, E3 +13718.973}
SPL {X  -156.808, Y  +353.900, Z    +0.000, E1   +73.180, E3 +13731.577}
SPL {X  -154.539, Y  +344.254, Z    +0.000, E1   +72.827, E3 +13741.115}
ENDSPLINE

SPLINE
SPL {X  -157.258, Y  +356.206, Z    +0.000, E1   +70.434, E3 +13755.687}
ENDSPLINE

SPLINE
SPL {X  -150.342, Y  +330.952, Z    +0.000, E1   +71.154, E3 +13767.359}
SPL {X  -141.358, Y  +310.748, Z    +0.000, E1   +71.233, E3 +13780.065}
SPL {X  -134.330, Y  +298.778, Z    +0.000, E1   +70.323, E3 +13793.912}
SPL {X  -128.957, Y  +290.989, Z    +0.000, E1   +69.528, E3 +13803.277}
SPL {X  -124.846, Y  +285.632, Z    +0.000, E1   +68.906, E3 +13809.741}
SPL {X  -121.783, Y  +281.927, Z    +0.000, E1   +68.403, E3 +13814.173}
SPL {X   -79.219, Y  +246.688, Z    +0.000, E1   +55.887, E3 +13935.679}
ENDSPLINE

SPLINE
SPL {X  -125.038, Y  +285.873, Z    +0.000, E1   +53.023, E3 +14112.720}
SPL {X  -149.949, Y  +329.886, Z    +0.000, E1   +41.515, E3 +14134.286}
SPL {X  -157.246, Y  +356.141, Z    +0.000, E1   +27.282, E3 +14139.342}
SPL {X  -159.525, Y  +373.376, Z    +0.000, E1   +13.812, E3 +14140.999}
SPL {X  -160.000, Y  +387.264, Z    +0.000, E1    +0.544, E3 +14141.457}
SPL {X  -160.000, Y  +390.384, Z    +0.000, E1    -6.008, E3 +14141.494}
SPL {X  -160.000, Y  +395.752, Z    +0.000, E1   -19.038, E3 +14141.688}
SPL {X  -160.000, Y  +404.289, Z    +0.000, E1   -38.292, E3 +14142.356}
SPL {X  -160.000, Y  +418.681, Z    +0.000, E1   -56.949, E3 +14144.546}
SPL {X  -160.000, Y  +471.977, Z    +0.000, E1   -70.792, E3 +14161.065}
SPL {X  -159.977, Y  +677.138, Z    +0.000, E1   -73.665, E3 +14257.556}
SPL {X  -157.805, Y  +700.810, Z    +0.000, E1   -73.511, E3 +14274.387}
SPL {X  -152.242, Y  +723.618, Z    +0.000, E1   -72.940, E3 +14294.299}
SPL {X  -145.929, Y  +740.010, Z    +0.000, E1   -72.229, E3 +14310.771}
SPL {X  -139.114, Y  +753.439, Z    +0.000, E1   -71.436, E3 +14325.409}
SPL {X  -132.333, Y  +764.333, Z    +0.000, E1   -70.535, E3 +14338.033}
SPL {X  -125.486, Y  +773.664, Z    +0.000, E1   -69.598, E3 +14349.007}
SPL {X  -121.321, Y  +778.713, Z    +0.000, E1   -68.872, E3 +14355.017}
SPL {X   -77.337, Y  +814.468, Z    +0.000, E1   -56.377, E3 +14473.649}
ENDSPLINE

SPLINE
SPL {X  -134.727, Y  +760.706, Z    +0.000, E1   -50.460, E3 +14661.881}
SPL {X  -155.580, Y  +711.748, Z    +0.000, E1   -32.084, E3 +14678.795}
SPL {X  -159.445, Y  +687.715, Z    +0.000, E1   -14.660, E3 +14681.642}
SPL {X  -159.995, Y  +675.725, Z    +0.000, E1    -3.424, E3 +14682.153}
SPL {X  -160.000, Y  +671.714, Z    +0.000, E1    +0.835, E3 +14682.193}
SPL {X  -160.000, Y  +663.084, Z    +0.000, E1   +21.134, E3 +14682.518}
SPL {X  -160.000, Y  +650.910, Z    +0.000, E1   +46.005, E3 +14683.671}
SPL {X  -160.000, Y  +634.843, Z    +0.000, E1   +61.273, E3 +14686.348}
SPL {X  -160.000, Y  +578.679, Z    +0.000, E1   +71.665, E3 +14704.182}
SPL {X  -160.000, Y  +387.528, Z    +0.000, E1   +73.487, E3 +14796.994}
SPL {X  -159.218, Y  +369.903, Z    +0.000, E1   +73.425, E3 +14808.862}
SPL {X  -156.808, Y  +353.900, Z    +0.000, E1   +73.180, E3 +14821.465}
SPL {X  -154.539, Y  +344.254, Z    +0.000, E1   +72.827, E3 +14831.003}
ENDSPLINE

SPLINE
SPL {X  -157.258, Y  +356.206, Z    +0.000, E1   +70.434, E3 +14845.575}
ENDSPLINE

SPLINE
SPL {X  -150.342, Y  +330.952, Z    +0.000, E1   +71.154, E3 +14857.247}
SPL {X  -141.358, Y  +310.748, Z    +0.000, E1   +71.233, E3 +14869.953}
SPL {X  -134.330, Y  +298.778, Z    +0.000, E1   +70.323, E3 +14883.800}
SPL {X  -128.957, Y  +290.989, Z    +0.000, E1   +69.528, E3 +14893.166}
SPL {X  -124.846, Y  +285.632, Z    +0.000, E1   +68.906, E3 +14899.629}
SPL {X  -121.783, Y  +281.927, Z    +0.000, E1   +68.403, E3 +14904.061}
SPL {X   -79.219, Y  +246.688, Z    +0.000, E1   +55.887, E3 +15025.567}
ENDSPLINE

SPLINE
SPL {X  -125.038, Y  +285.873, Z    +0.000, E1   +53.023, E3 +15202.608}
SPL {X  -149.949, Y  +329.886, Z    +0.000, E1   +41.515, E3 +15224.174}
SPL {X  -157.246, Y  +356.141, Z    +0.000, E1   +27.282, E3 +15229.230}
SPL {X  -159.525, Y  +373.376, Z    +0.000, E1   +13.812, E3 +15230.887}
SPL {X  -160.000, Y  +387.264, Z    +0.000, E1    +0.544, E3 +15231.345}
SPL {X  -160.000, Y  +390.384, Z    +0.000, E1    -6.008, E3 +15231.382}
SPL {X  -160.000, Y  +395.752, Z    +0.000, E1   -19.038, E3 +15231.576}
SPL {X  -160.000, Y  +404.289, Z    +0.000, E1   -38.292, E3 +15232.244}
SPL {X  -160.000, Y  +418.681, Z    +0.000, E1   -56.949, E3 +15234.434}
SPL {X  -160.000, Y  +471.977, Z    +0.000, E1   -70.792, E3 +15250.953}
SPL {X  -159.977, Y  +677.138, Z    +0.000, E1   -73.665, E3 +15347.444}
SPL {X  -157.805, Y  +700.810, Z    +0.000, E1   -73.511, E3 +15364.275}
SPL {X  -152.242, Y  +723.618, Z    +0.000, E1   -72.940, E3 +15384.187}
SPL {X  -145.929, Y  +740.010, Z    +0.000, E1   -72.229, E3 +15400.659}
SPL {X  -139.114, Y  +753.439, Z    +0.000, E1   -71.436, E3 +15415.297}
SPL {X  -132.333, Y  +764.333, Z    +0.000, E1   -70.535, E3 +15427.921}
SPL {X  -125.486, Y  +773.664, Z    +0.000, E1   -69.598, E3 +15438.895}
SPL {X  -121.321, Y  +778.713, Z    +0.000, E1   -68.872, E3 +15444.905}
SPL {X   -77.337, Y  +814.468, Z    +0.000, E1   -56.377, E3 +15563.537}
ENDSPLINE

SPLINE
SPL {X  -134.727, Y  +760.706, Z    +0.000, E1   -50.460, E3 +15751.769}
SPL {X  -155.580, Y  +711.748, Z    +0.000, E1   -32.084, E3 +15768.683}
SPL {X  -159.445, Y  +687.715, Z    +0.000, E1   -14.660, E3 +15771.530}
SPL {X  -159.995, Y  +675.725, Z    +0.000, E1    -3.424, E3 +15772.041}
SPL {X  -160.000, Y  +671.714, Z    +0.000, E1    +0.835, E3 +15772.081}
SPL {X  -160.000, Y  +663.084, Z    +0.000, E1   +21.134, E3 +15772.406}
SPL {X  -160.000, Y  +650.910, Z    +0.000, E1   +46.005, E3 +15773.559}
SPL {X  -160.000, Y  +634.843, Z    +0.000, E1   +61.273, E3 +15776.236}
SPL {X  -160.000, Y  +578.679, Z    +0.000, E1   +71.665, E3 +15794.070}
SPL {X  -160.000, Y  +387.528, Z    +0.000, E1   +73.487, E3 +15886.882}
SPL {X  -159.218, Y  +369.903, Z    +0.000, E1   +73.425, E3 +15898.750}
SPL {X  -156.808, Y  +353.900, Z    +0.000, E1   +73.180, E3 +15911.353}
SPL {X  -154.539, Y  +344.254, Z    +0.000, E1   +72.827, E3 +15920.891}
ENDSPLINE

SPLINE
SPL {X  -157.258, Y  +356.206, Z    +0.000, E1   +70.434, E3 +15935.463}
ENDSPLINE

SPLINE
SPL {X  -150.342, Y  +330.952, Z    +0.000, E1   +71.154, E3 +15947.135}
SPL {X  -141.358, Y  +310.748, Z    +0.000, E1   +71.233, E3 +15959.841}
SPL {X  -134.330, Y  +298.778, Z    +0.000, E1   +70.323, E3 +15973.688}
SPL {X  -128.957, Y  +290.989, Z    +0.000, E1   +69.528, E3 +15983.054}
SPL {X  -124.846, Y  +285.632, Z    +0.000, E1   +68.906, E3 +15989.517}
SPL {X  -121.783, Y  +281.927, Z    +0.000, E1   +68.403, E3 +15993.949}
SPL {X   -79.219, Y  +246.688, Z    +0.000, E1   +55.887, E3 +16115.455}
ENDSPLINE

SPLINE
SPL {X  -125.038, Y  +285.873, Z    +0.000, E1   +53.023, E3 +16292.497}
SPL {X  -149.949, Y  +329.886, Z    +0.000, E1   +41.515, E3 +16314.062}
SPL {X  -157.246, Y  +356.141, Z    +0.000, E1   +27.282, E3 +16319.118}
SPL {X  -159.525, Y  +373.376, Z    +0.000, E1   +13.812, E3 +16320.775}
SPL {X  -160.000, Y  +387.264, Z    +0.000, E1    +0.544, E3 +16321.233}
SPL {X  -160.000, Y  +390.384, Z    +0.000, E1    -6.008, E3 +16321.270}
SPL {X  -160.000, Y  +395.752, Z    +0.000, E1   -19.038, E3 +16321.464}
SPL {X  -160.000, Y  +404.289, Z    +0.000, E1   -38.292, E3 +16322.132}
SPL {X  -160.000, Y  +418.681, Z    +0.000, E1   -56.949, E3 +16324.322}
SPL {X  -160.000, Y  +471.977, Z    +0.000, E1   -70.792, E3 +16340.841}
SPL {X  -159.977, Y  +677.138, Z    +0.000, E1   -73.665, E3 +16437.332}
SPL {X  -157.805, Y  +700.810, Z    +0.000, E1   -73.511, E3 +16454.163}
SPL {X  -152.242, Y  +723.618, Z    +0.000, E1   -72.940, E3 +16474.076}
SPL {X  -145.929, Y  +740.010, Z    +0.000, E1   -72.229, E3 +16490.547}
SPL {X  -139.114, Y  +753.439, Z    +0.000, E1   -71.436, E3 +16505.186}
SPL {X  -132.333, Y  +764.333, Z    +0.000, E1   -70.535, E3 +16517.809}
SPL {X  -125.486, Y  +773.664, Z    +0.000, E1   -69.598, E3 +16528.784}
SPL {X  -121.321, Y  +778.713, Z    +0.000, E1   -68.872, E3 +16534.794}
SPL {X   -77.337, Y  +814.468, Z    +0.000, E1   -56.377, E3 +16653.425}
ENDSPLINE

SPLINE
SPL {X  -134.727, Y  +760.706, Z    +0.000, E1   -50.460, E3 +16841.657}
SPL {X  -155.580, Y  +711.748, Z    +0.000, E1   -32.084, E3 +16858.571}
SPL {X  -159.445, Y  +687.715, Z    +0.000, E1   -14.660, E3 +16861.418}
SPL {X  -159.995, Y  +675.725, Z    +0.000, E1    -3.424, E3 +16861.929}
SPL {X  -160.000, Y  +671.714, Z    +0.000, E1    +0.835, E3 +16861.969}
SPL {X  -160.000, Y  +663.084, Z    +0.000, E1   +21.134, E3 +16862.294}
SPL {X  -160.000, Y  +650.910, Z    +0.000, E1   +46.005, E3 +16863.447}
SPL {X  -160.000, Y  +634.843, Z    +0.000, E1   +61.273, E3 +16866.124}
SPL {X  -160.000, Y  +578.679, Z    +0.000, E1   +71.665, E3 +16883.958}
SPL {X  -160.000, Y  +387.528, Z    +0.000, E1   +73.487, E3 +16976.770}
SPL {X  -159.218, Y  +369.903, Z    +0.000, E1   +73.425, E3 +16988.638}
SPL {X  -156.808, Y  +353.900, Z    +0.000, E1   +73.180, E3 +17001.241}
SPL {X  -154.539, Y  +344.254, Z    +0.000, E1   +72.827, E3 +17010.779}
ENDSPLINE

SPLINE
SPL {X  -157.258, Y  +356.206, Z    +0.000, E1   +70.434, E3 +17025.351}
ENDSPLINE

SPLINE
SPL {X  -150.342, Y  +330.952, Z    +0.000, E1   +71.154, E3 +17037.023}
SPL {X  -141.358, Y  +310.748, Z    +0.000, E1   +71.233, E3 +17049.729}
SPL {X  -134.330, Y  +298.778, Z    +0.000, E1   +70.323, E3 +17063.576}
SPL {X  -128.957, Y  +290.989, Z    +0.000, E1   +69.528, E3 +17072.942}
SPL {X  -124.846, Y  +285.632, Z    +0.000, E1   +68.906, E3 +17079.405}
SPL {X  -121.783, Y  +281.927, Z    +0.000, E1   +68.403, E3 +17083.837}
SPL {X   -79.219, Y  +246.688, Z    +0.000, E1   +55.887, E3 +17205.343}
ENDSPLINE

SPLINE
SPL {X  -125.038, Y  +285.873, Z    +0.000, E1   +53.023, E3 +17382.385}
SPL {X  -149.949, Y  +329.886, Z    +0.000, E1   +41.515, E3 +17403.950}
SPL {X  -157.246, Y  +356.141, Z    +0.000, E1   +27.282, E3 +17409.006}
SPL {X  -159.525, Y  +373.376, Z    +0.000, E1   +13.812, E3 +17410.663}
SPL {X  -160.000, Y  +387.264, Z    +0.000, E1    +0.544, E3 +17411.121}
SPL {X  -160.000, Y  +390.384, Z    +0.000, E1    -6.008, E3 +17411.158}
SPL {X  -160.000, Y  +395.752, Z    +0.000, E1   -19.038, E3 +17411.352}
SPL {X  -160.000, Y  +404.289, Z    +0.000, E1   -38.292, E3 +17412.020}
SPL {X  -160.000, Y  +418.681, Z    +0.000, E1   -56.949, E3 +17414.210}
SPL {X  -160.000, Y  +458.961, Z    +0.000, E1   -69.778, E3 +17425.806}
SPL {X  -160.000, Y  +485.343, Z    +0.000, E1   -71.539, E3 +17435.792}
SPL {X  -159.977, Y  +677.138, Z    +0.000, E1   -73.665, E3 +17527.220}
SPL {X  -157.805, Y  +700.810, Z    +0.000, E1   -73.511, E3 +17544.051}
SPL {X  -152.242, Y  +723.618, Z    +0.000, E1   -72.940, E3 +17563.964}
SPL {X  -145.929, Y  +740.010, Z    +0.000, E1   -72.229, E3 +17580.435}
SPL {X  -139.114, Y  +753.439, Z    +0.000, E1   -71.436, E3 +17595.074}
SPL {X  -132.333, Y  +764.333, Z    +0.000, E1   -70.535, E3 +17607.697}
SPL {X  -125.486, Y  +773.664, Z    +0.000, E1   -69.598, E3 +17618.672}
SPL {X  -121.321, Y  +778.713, Z    +0.000, E1   -68.872, E3 +17624.682}
SPL {X   -77.337, Y  +814.468, Z    +0.000, E1   -56.377, E3 +17743.313}
ENDSPLINE

SPLINE
SPL {X  -134.727, Y  +760.706, Z    +0.000, E1   -50.460, E3 +17931.545}
SPL {X  -155.580, Y  +711.748, Z    +0.000, E1   -32.084, E3 +17948.459}
SPL {X  -159.445, Y  +687.715, Z    +0.000, E1   -14.660, E3 +17951.306}
SPL {X  -159.995, Y  +675.725, Z    +0.000, E1    -3.424, E3 +17951.817}
SPL {X  -160.000, Y  +671.714, Z    +0.000, E1    +0.835, E3 +17951.857}
SPL {X  -160.000, Y  +663.084, Z    +0.000, E1   +21.134, E3 +17952.182}
SPL {X  -160.000, Y  +650.910, Z    +0.000, E1   +46.005, E3 +17953.335}
SPL {X  -160.000, Y  +634.843, Z    +0.000, E1   +61.273, E3 +17956.012}
SPL {X  -160.000, Y  +578.679, Z    +0.000, E1   +71.665, E3 +17973.846}
SPL {X  -160.000, Y  +387.528, Z    +0.000, E1   +73.487, E3 +18066.658}
SPL {X  -159.218, Y  +369.903, Z    +0.000, E1   +73.425, E3 +18078.526}
SPL {X  -156.808, Y  +353.900, Z    +0.000, E1   +73.180, E3 +18091.129}
SPL {X  -154.539, Y  +344.254, Z    +0.000, E1   +72.827, E3 +18100.667}
ENDSPLINE

SPLINE
SPL {X  -157.258, Y  +356.206, Z    +0.000, E1   +70.434, E3 +18115.239}
ENDSPLINE

SPLINE
SPL {X  -150.342, Y  +330.952, Z    +0.000, E1   +71.154, E3 +18126.911}
SPL {X  -141.358, Y  +310.748, Z    +0.000, E1   +71.233, E3 +18139.617}
SPL {X  -134.330, Y  +298.778, Z    +0.000, E1   +70.323, E3 +18153.464}
SPL {X  -128.957, Y  +290.989, Z    +0.000, E1   +69.528, E3 +18162.830}
SPL {X  -124.846, Y  +285.632, Z    +0.000, E1   +68.906, E3 +18169.293}
SPL {X  -121.783, Y  +281.927, Z    +0.000, E1   +68.403, E3 +18173.725}
SPL {X   -79.219, Y  +246.688, Z    +0.000, E1   +55.887, E3 +18295.231}
ENDSPLINE

SPLINE
SPL {X  -125.038, Y  +285.873, Z    +0.000, E1   +53.023, E3 +18472.273}
SPL {X  -149.949, Y  +329.886, Z    +0.000, E1   +41.515, E3 +18493.838}
SPL {X  -157.246, Y  +356.141, Z    +0.000, E1   +27.282, E3 +18498.894}
SPL {X  -159.525, Y  +373.376, Z    +0.000, E1   +13.812, E3 +18500.551}
SPL {X  -160.000, Y  +387.264, Z    +0.000, E1    +0.544, E3 +18501.009}
SPL {X  -160.000, Y  +390.384, Z    +0.000, E1    -6.008, E3 +18501.046}
SPL {X  -160.000, Y  +395.752, Z    +0.000, E1   -19.038, E3 +18501.240}
SPL {X  -160.000, Y  +404.289, Z    +0.000, E1   -38.292, E3 +18501.908}
SPL {X  -160.000, Y  +418.681, Z    +0.000, E1   -56.949, E3 +18504.098}
SPL {X  -160.000, Y  +458.961, Z    +0.000, E1   -69.778, E3 +18515.694}
SPL {X  -160.000, Y  +485.343, Z    +0.000, E1   -71.539, E3 +18525.680}
SPL {X  -159.977, Y  +677.138, Z    +0.000, E1   -73.665, E3 +18617.109}
SPL {X  -157.805, Y  +700.810, Z    +0.000, E1   -73.511, E3 +18633.939}
SPL {X  -152.242, Y  +723.618, Z    +0.000, E1   -72.940, E3 +18653.852}
SPL {X  -145.929, Y  +740.010, Z    +0.000, E1   -72.229, E3 +18670.323}
SPL {X  -139.114, Y  +753.439, Z    +0.000, E1   -71.436, E3 +18684.962}
SPL {X  -132.333, Y  +764.333, Z    +0.000, E1   -70.535, E3 +18697.585}
SPL {X  -125.486, Y  +773.664, Z    +0.000, E1   -69.598, E3 +18708.560}
SPL {X  -121.321, Y  +778.713, Z    +0.000, E1   -68.872, E3 +18714.570}
SPL {X   -77.337, Y  +814.468, Z    +0.000, E1   -56.377, E3 +18833.201}
ENDSPLINE

SPLINE
SPL {X  -134.727, Y  +760.706, Z    +0.000, E1   -50.460, E3 +19021.433}
SPL {X  -155.580, Y  +711.748, Z    +0.000, E1   -32.084, E3 +19038.347}
SPL {X  -159.445, Y  +687.715, Z    +0.000, E1   -14.660, E3 +19041.194}
SPL {X  -159.995, Y  +675.725, Z    +0.000, E1    -3.424, E3 +19041.705}
SPL {X  -160.000, Y  +671.714, Z    +0.000, E1    +0.835, E3 +19041.745}
SPL {X  -160.000, Y  +663.084, Z    +0.000, E1   +21.134, E3 +19042.070}
SPL {X  -160.000, Y  +650.910, Z    +0.000, E1   +46.005, E3 +19043.223}
SPL {X  -160.000, Y  +634.843, Z    +0.000, E1   +61.273, E3 +19045.900}
SPL {X  -160.000, Y  +578.679, Z    +0.000, E1   +71.665, E3 +19063.734}
SPL {X  -160.000, Y  +387.528, Z    +0.000, E1   +73.487, E3 +19156.546}
SPL {X  -159.218, Y  +369.903, Z    +0.000, E1   +73.425, E3 +19168.414}
SPL {X  -156.808, Y  +353.900, Z    +0.000, E1   +73.180, E3 +19181.017}
SPL {X  -154.539, Y  +344.254, Z    +0.000, E1   +72.827, E3 +19190.555}
ENDSPLINE

SPLINE
SPL {X  -157.258, Y  +356.206, Z    +0.000, E1   +70.434, E3 +19205.127}
ENDSPLINE

SPLINE
SPL {X  -150.342, Y  +330.952, Z    +0.000, E1   +71.154, E3 +19216.800}
SPL {X  -141.358, Y  +310.748, Z    +0.000, E1   +71.233, E3 +19229.505}
SPL {X  -134.330, Y  +298.778, Z    +0.000, E1   +70.323, E3 +19243.352}
SPL {X  -128.957, Y  +290.989, Z    +0.000, E1   +69.528, E3 +19252.718}
SPL {X  -124.846, Y  +285.632, Z    +0.000, E1   +68.906, E3 +19259.181}
SPL {X  -121.783, Y  +281.927, Z    +0.000, E1   +68.403, E3 +19263.613}
SPL {X   -79.219, Y  +246.688, Z    +0.000, E1   +55.887, E3 +19385.120}
ENDSPLINE

SPLINE
SPL {X  -125.038, Y  +285.873, Z    +0.000, E1   +53.023, E3 +19562.161}
SPL {X  -149.949, Y  +329.886, Z    +0.000, E1   +41.515, E3 +19583.726}
SPL {X  -157.246, Y  +356.141, Z    +0.000, E1   +27.282, E3 +19588.782}
SPL {X  -159.525, Y  +373.376, Z    +0.000, E1   +13.812, E3 +19590.439}
SPL {X  -160.000, Y  +387.264, Z    +0.000, E1    +0.544, E3 +19590.897}
SPL {X  -160.000, Y  +390.384, Z    +0.000, E1    -6.008, E3 +19590.934}
SPL {X  -160.000, Y  +395.752, Z    +0.000, E1   -19.038, E3 +19591.128}
SPL {X  -160.000, Y  +404.289, Z    +0.000, E1   -38.292, E3 +19591.796}
SPL {X  -160.000, Y  +418.681, Z    +0.000, E1   -56.949, E3 +19593.986}
SPL {X  -160.000, Y  +471.977, Z    +0.000, E1   -70.792, E3 +19610.505}
SPL {X  -159.977, Y  +677.138, Z    +0.000, E1   -73.665, E3 +19706.997}
SPL {X  -157.805, Y  +700.810, Z    +0.000, E1   -73.511, E3 +19723.827}
SPL {X  -152.242, Y  +723.618, Z    +0.000, E1   -72.940, E3 +19743.740}
SPL {X  -145.929, Y  +740.010, Z    +0.000, E1   -72.229, E3 +19760.211}
SPL {X  -139.114, Y  +753.439, Z    +0.000, E1   -71.436, E3 +19774.850}
SPL {X  -132.333, Y  +764.333, Z    +0.000, E1   -70.535, E3 +19787.473}
SPL {X  -125.486, Y  +773.664, Z    +0.000, E1   -69.598, E3 +19798.448}
SPL {X  -121.321, Y  +778.713, Z    +0.000, E1   -68.872, E3 +19804.458}
SPL {X   -77.337, Y  +814.468, Z    +0.000, E1   -56.377, E3 +19923.089}
ENDSPLINE

SPLINE
SPL {X  -134.727, Y  +760.706, Z    +0.000, E1   -50.460, E3 +20111.321}
SPL {X  -155.580, Y  +711.748, Z    +0.000, E1   -32.084, E3 +20128.235}
SPL {X  -159.445, Y  +687.715, Z    +0.000, E1   -14.660, E3 +20131.082}
SPL {X  -159.995, Y  +675.725, Z    +0.000, E1    -3.424, E3 +20131.593}
SPL {X  -160.000, Y  +671.714, Z    +0.000, E1    +0.835, E3 +20131.633}
SPL {X  -160.000, Y  +663.084, Z    +0.000, E1   +21.134, E3 +20131.958}
SPL {X  -160.000, Y  +650.910, Z    +0.000, E1   +46.005, E3 +20133.111}
SPL {X  -160.000, Y  +634.843, Z    +0.000, E1   +61.273, E3 +20135.788}
SPL {X  -160.000, Y  +578.679, Z    +0.000, E1   +71.665, E3 +20153.622}
SPL {X  -160.000, Y  +387.528, Z    +0.000, E1   +73.487, E3 +20246.434}
SPL {X  -159.218, Y  +369.903, Z    +0.000, E1   +73.425, E3 +20258.302}
SPL {X  -156.808, Y  +353.900, Z    +0.000, E1   +73.180, E3 +20270.905}
SPL {X  -154.539, Y  +344.254, Z    +0.000, E1   +72.827, E3 +20280.443}
ENDSPLINE

SPLINE
SPL {X  -157.258, Y  +356.206, Z    +0.000, E1   +70.434, E3 +20295.015}
ENDSPLINE

SPLINE
SPL {X  -150.342, Y  +330.952, Z    +0.000, E1   +71.154, E3 +20306.688}
SPL {X  -141.358, Y  +310.748, Z    +0.000, E1   +71.233, E3 +20319.393}
SPL {X  -134.330, Y  +298.778, Z    +0.000, E1   +70.323, E3 +20333.241}
SPL {X  -128.957, Y  +290.989, Z    +0.000, E1   +69.528, E3 +20342.606}
SPL {X  -124.846, Y  +285.632, Z    +0.000, E1   +68.906, E3 +20349.069}
SPL {X  -121.783, Y  +281.927, Z    +0.000, E1   +68.403, E3 +20353.501}
SPL {X   -79.219, Y  +246.688, Z    +0.000, E1   +55.887, E3 +20475.008}
ENDSPLINE

SPLINE
SPL {X  -125.038, Y  +285.873, Z    +0.000, E1   +53.023, E3 +20652.049}
SPL {X  -149.949, Y  +329.886, Z    +0.000, E1   +41.515, E3 +20673.614}
SPL {X  -157.246, Y  +356.141, Z    +0.000, E1   +27.282, E3 +20678.670}
SPL {X  -159.525, Y  +373.376, Z    +0.000, E1   +13.812, E3 +20680.327}
SPL {X  -160.000, Y  +387.264, Z    +0.000, E1    +0.544, E3 +20680.785}
SPL {X  -160.000, Y  +390.384, Z    +0.000, E1    -6.008, E3 +20680.822}
SPL {X  -160.000, Y  +395.752, Z    +0.000, E1   -19.038, E3 +20681.016}
SPL {X  -160.000, Y  +404.289, Z    +0.000, E1   -38.292, E3 +20681.684}
SPL {X  -160.000, Y  +418.681, Z    +0.000, E1   -56.949, E3 +20683.874}
SPL {X  -160.000, Y  +471.977, Z    +0.000, E1   -70.792, E3 +20700.393}
SPL {X  -159.977, Y  +677.138, Z    +0.000, E1   -73.665, E3 +20796.885}
SPL {X  -157.805, Y  +700.810, Z    +0.000, E1   -73.511, E3 +20813.715}
SPL {X  -152.242, Y  +723.618, Z    +0.000, E1   -72.940, E3 +20833.628}
SPL {X  -145.929, Y  +740.010, Z    +0.000, E1   -72.229, E3 +20850.099}
SPL {X  -139.114, Y  +753.439, Z    +0.000, E1   -71.436, E3 +20864.738}
SPL {X  -132.333, Y  +764.333, Z    +0.000, E1   -70.535, E3 +20877.362}
SPL {X  -125.486, Y  +773.664, Z    +0.000, E1   -69.598, E3 +20888.336}
SPL {X  -121.321, Y  +778.713, Z    +0.000, E1   -68.872, E3 +20894.346}
SPL {X   -77.337, Y  +814.468, Z    +0.000, E1   -56.377, E3 +21012.977}
ENDSPLINE

SPLINE
SPL {X  -134.727, Y  +760.706, Z    +0.000, E1   -50.460, E3 +21201.209}
SPL {X  -155.580, Y  +711.748, Z    +0.000, E1   -32.084, E3 +21218.123}
SPL {X  -159.445, Y  +687.715, Z    +0.000, E1   -14.660, E3 +21220.970}
SPL {X  -159.995, Y  +675.725, Z    +0.000, E1    -3.424, E3 +21221.481}
SPL {X  -160.000, Y  +671.714, Z    +0.000, E1    +0.835, E3 +21221.521}
SPL {X  -160.000, Y  +663.084, Z    +0.000, E1   +21.134, E3 +21221.846}
SPL {X  -160.000, Y  +650.910, Z    +0.000, E1   +46.005, E3 +21223.000}
SPL {X  -160.000, Y  +634.843, Z    +0.000, E1   +61.273, E3 +21225.676}
SPL {X  -160.000, Y  +578.679, Z    +0.000, E1   +71.665, E3 +21243.510}
SPL {X  -160.000, Y  +387.528, Z    +0.000, E1   +73.487, E3 +21336.323}
SPL {X  -159.218, Y  +369.903, Z    +0.000, E1   +73.425, E3 +21348.190}
SPL {X  -156.808, Y  +353.900, Z    +0.000, E1   +73.180, E3 +21360.793}
SPL {X  -154.539, Y  +344.254, Z    +0.000, E1   +72.827, E3 +21370.331}
ENDSPLINE

SPLINE
SPL {X  -157.258, Y  +356.206, Z    +0.000, E1   +70.434, E3 +21384.903}
ENDSPLINE

SPLINE
SPL {X  -150.342, Y  +330.952, Z    +0.000, E1   +71.154, E3 +21396.576}
SPL {X  -141.358, Y  +310.748, Z    +0.000, E1   +71.233, E3 +21409.281}
SPL {X  -134.330, Y  +298.778, Z    +0.000, E1   +70.323, E3 +21423.129}
SPL {X  -128.957, Y  +290.989, Z    +0.000, E1   +69.528, E3 +21432.494}
SPL {X  -124.846, Y  +285.632, Z    +0.000, E1   +68.906, E3 +21438.957}
SPL {X  -121.783, Y  +281.927, Z    +0.000, E1   +68.403, E3 +21443.389}
SPL {X   -79.219, Y  +246.688, Z    +0.000, E1   +55.887, E3 +21564.896}
ENDSPLINE

SPLINE
SPL {X  -125.038, Y  +285.873, Z    +0.000, E1   +53.023, E3 +21741.937}
SPL {X  -149.949, Y  +329.886, Z    +0.000, E1   +41.515, E3 +21763.502}
SPL {X  -157.246, Y  +356.141, Z    +0.000, E1   +27.282, E3 +21768.558}
SPL {X  -159.525, Y  +373.376, Z    +0.000, E1   +13.812, E3 +21770.216}
SPL {X  -160.000, Y  +387.264, Z    +0.000, E1    +0.544, E3 +21770.673}
SPL {X  -160.000, Y  +390.384, Z    +0.000, E1    -6.008, E3 +21770.710}
SPL {X  -160.000, Y  +395.752, Z    +0.000, E1   -19.038, E3 +21770.904}
SPL {X  -160.000, Y  +404.289, Z    +0.000, E1   -38.292, E3 +21771.573}
SPL {X  -160.000, Y  +418.681, Z    +0.000, E1   -56.949, E3 +21773.762}
SPL {X  -160.000, Y  +471.977, Z    +0.000, E1   -70.792, E3 +21790.282}
SPL {X  -159.977, Y  +677.138, Z    +0.000, E1   -73.665, E3 +21886.773}
SPL {X  -157.805, Y  +700.810, Z    +0.000, E1   -73.511, E3 +21903.603}
SPL {X  -152.242, Y  +723.618, Z    +0.000, E1   -72.940, E3 +21923.516}
SPL {X  -145.929, Y  +740.010, Z    +0.000, E1   -72.229, E3 +21939.987}
SPL {X  -139.114, Y  +753.439, Z    +0.000, E1   -71.436, E3 +21954.626}
SPL {X  -132.333, Y  +764.333, Z    +0.000, E1   -70.535, E3 +21967.250}
SPL {X  -125.486, Y  +773.664, Z    +0.000, E1   -69.598, E3 +21978.224}
SPL {X  -121.321, Y  +778.713, Z    +0.000, E1   -68.872, E3 +21984.234}
SPL {X   -77.337, Y  +814.468, Z    +0.000, E1   -56.377, E3 +22102.865}
ENDSPLINE

SPLINE
SPL {X  -134.727, Y  +760.706, Z    +0.000, E1   -50.460, E3 +22291.097}
SPL {X  -155.580, Y  +711.748, Z    +0.000, E1   -32.084, E3 +22308.012}
SPL {X  -159.445, Y  +687.715, Z    +0.000, E1   -14.660, E3 +22310.858}
SPL {X  -159.995, Y  +675.725, Z    +0.000, E1    -3.424, E3 +22311.369}
SPL {X  -160.000, Y  +671.714, Z    +0.000, E1    +0.835, E3 +22311.410}
SPL {X  -160.000, Y  +663.084, Z    +0.000, E1   +21.134, E3 +22311.734}
SPL {X  -160.000, Y  +650.910, Z    +0.000, E1   +46.005, E3 +22312.888}
SPL {X  -160.000, Y  +634.843, Z    +0.000, E1   +61.273, E3 +22315.564}
SPL {X  -160.000, Y  +578.679, Z    +0.000, E1   +71.665, E3 +22333.398}
SPL {X  -160.000, Y  +387.528, Z    +0.000, E1   +73.487, E3 +22426.211}
SPL {X  -159.218, Y  +369.903, Z    +0.000, E1   +73.425, E3 +22438.078}
SPL {X  -156.808, Y  +353.900, Z    +0.000, E1   +73.180, E3 +22450.682}
SPL {X  -154.539, Y  +344.254, Z    +0.000, E1   +72.827, E3 +22460.219}
ENDSPLINE

SPLINE
SPL {X  -157.258, Y  +356.206, Z    +0.000, E1   +70.434, E3 +22474.791}
ENDSPLINE

SPLINE
SPL {X  -150.342, Y  +330.952, Z    +0.000, E1   +71.154, E3 +22486.464}
SPL {X  -141.358, Y  +310.748, Z    +0.000, E1   +71.233, E3 +22499.169}
SPL {X  -134.330, Y  +298.778, Z    +0.000, E1   +70.323, E3 +22513.017}
SPL {X  -128.957, Y  +290.989, Z    +0.000, E1   +69.528, E3 +22522.382}
SPL {X  -124.846, Y  +285.632, Z    +0.000, E1   +68.906, E3 +22528.845}
SPL {X  -121.783, Y  +281.927, Z    +0.000, E1   +68.403, E3 +22533.277}
SPL {X   -79.219, Y  +246.688, Z    +0.000, E1   +55.887, E3 +22654.784}
ENDSPLINE

SPLINE
SPL {X  -125.038, Y  +285.873, Z    +0.000, E1   +53.023, E3 +22831.825}
SPL {X  -149.949, Y  +329.886, Z    +0.000, E1   +41.515, E3 +22853.390}
SPL {X  -157.246, Y  +356.141, Z    +0.000, E1   +27.282, E3 +22858.446}
SPL {X  -159.525, Y  +373.376, Z    +0.000, E1   +13.812, E3 +22860.104}
SPL {X  -160.000, Y  +387.264, Z    +0.000, E1    +0.544, E3 +22860.561}
SPL {X  -160.000, Y  +390.384, Z    +0.000, E1    -6.008, E3 +22860.598}
SPL {X  -160.000, Y  +395.752, Z    +0.000, E1   -19.038, E3 +22860.792}
SPL {X  -160.000, Y  +404.289, Z    +0.000, E1   -38.292, E3 +22861.461}
SPL {X  -160.000, Y  +418.681, Z    +0.000, E1   -56.949, E3 +22863.650}
SPL {X  -160.000, Y  +471.977, Z    +0.000, E1   -70.792, E3 +22880.170}
SPL {X  -159.977, Y  +677.138, Z    +0.000, E1   -73.665, E3 +22976.661}
SPL {X  -157.805, Y  +700.810, Z    +0.000, E1   -73.511, E3 +22993.491}
SPL {X  -152.242, Y  +723.618, Z    +0.000, E1   -72.940, E3 +23013.404}
SPL {X  -145.929, Y  +740.010, Z    +0.000, E1   -72.229, E3 +23029.875}
SPL {X  -139.114, Y  +753.439, Z    +0.000, E1   -71.436, E3 +23044.514}
SPL {X  -132.333, Y  +764.333, Z    +0.000, E1   -70.535, E3 +23057.138}
SPL {X  -125.486, Y  +773.664, Z    +0.000, E1   -69.598, E3 +23068.112}
SPL {X  -121.321, Y  +778.713, Z    +0.000, E1   -68.872, E3 +23074.122}
SPL {X   -77.337, Y  +814.468, Z    +0.000, E1   -56.377, E3 +23192.753}
ENDSPLINE

SPLINE
SPL {X  -134.727, Y  +760.706, Z    +0.000, E1   -50.460, E3 +23380.985}
SPL {X  -155.580, Y  +711.748, Z    +0.000, E1   -32.084, E3 +23397.900}
SPL {X  -159.445, Y  +687.715, Z    +0.000, E1   -14.660, E3 +23400.746}
SPL {X  -159.995, Y  +675.725, Z    +0.000, E1    -3.424, E3 +23401.257}
SPL {X  -160.000, Y  +671.714, Z    +0.000, E1    +0.835, E3 +23401.298}
SPL {X  -160.000, Y  +663.084, Z    +0.000, E1   +21.134, E3 +23401.622}
SPL {X  -160.000, Y  +650.910, Z    +0.000, E1   +46.005, E3 +23402.776}
SPL {X  -160.000, Y  +634.843, Z    +0.000, E1   +61.273, E3 +23405.453}
SPL {X  -160.000, Y  +578.679, Z    +0.000, E1   +71.665, E3 +23423.286}
SPL {X  -160.000, Y  +387.528, Z    +0.000, E1   +73.487, E3 +23516.099}
SPL {X  -159.218, Y  +369.903, Z    +0.000, E1   +73.425, E3 +23527.966}
SPL {X  -156.808, Y  +353.900, Z    +0.000, E1   +73.180, E3 +23540.570}
SPL {X  -154.539, Y  +344.254, Z    +0.000, E1   +72.827, E3 +23550.107}
ENDSPLINE

SPLINE
SPL {X  -157.258, Y  +356.206, Z    +0.000, E1   +70.434, E3 +23564.679}
ENDSPLINE

SPLINE
SPL {X  -150.342, Y  +330.952, Z    +0.000, E1   +71.154, E3 +23576.352}
SPL {X  -141.358, Y  +310.748, Z    +0.000, E1   +71.233, E3 +23589.057}
SPL {X  -134.330, Y  +298.778, Z    +0.000, E1   +70.323, E3 +23602.905}
SPL {X  -128.957, Y  +290.989, Z    +0.000, E1   +69.528, E3 +23612.270}
SPL {X  -124.846, Y  +285.632, Z    +0.000, E1   +68.906, E3 +23618.733}
SPL {X  -121.783, Y  +281.927, Z    +0.000, E1   +68.403, E3 +23623.165}
SPL {X   -79.219, Y  +246.688, Z    +0.000, E1   +55.887, E3 +23744.672}
ENDSPLINE

SPLINE
SPL {X  -125.038, Y  +285.873, Z    +0.000, E1   +53.023, E3 +23921.713}
SPL {X  -149.949, Y  +329.886, Z    +0.000, E1   +41.515, E3 +23943.278}
SPL {X  -157.246, Y  +356.141, Z    +0.000, E1   +27.282, E3 +23948.335}
SPL {X  -159.525, Y  +373.376, Z    +0.000, E1   +13.812, E3 +23949.992}
SPL {X  -160.000, Y  +387.264, Z    +0.000, E1    +0.544, E3 +23950.449}
SPL {X  -160.000, Y  +390.384, Z    +0.000, E1    -6.008, E3 +23950.487}
SPL {X  -160.000, Y  +395.752, Z    +0.000, E1   -19.038, E3 +23950.680}
SPL {X  -160.000, Y  +404.289, Z    +0.000, E1   -38.292, E3 +23951.349}
SPL {X  -160.000, Y  +418.681, Z    +0.000, E1   -56.949, E3 +23953.538}
SPL {X  -160.000, Y  +471.977, Z    +0.000, E1   -70.792, E3 +23970.058}
SPL {X  -159.977, Y  +677.138, Z    +0.000, E1   -73.665, E3 +24066.549}
SPL {X  -157.805, Y  +700.810, Z    +0.000, E1   -73.511, E3 +24083.379}
SPL {X  -152.242, Y  +723.618, Z    +0.000, E1   -72.940, E3 +24103.292}
SPL {X  -145.929, Y  +740.010, Z    +0.000, E1   -72.229, E3 +24119.763}
SPL {X  -139.114, Y  +753.439, Z    +0.000, E1   -71.436, E3 +24134.402}
SPL {X  -132.333, Y  +764.333, Z    +0.000, E1   -70.535, E3 +24147.026}
SPL {X  -125.486, Y  +773.664, Z    +0.000, E1   -69.598, E3 +24158.000}
SPL {X  -121.321, Y  +778.713, Z    +0.000, E1   -68.872, E3 +24164.010}
SPL {X   -77.337, Y  +814.468, Z    +0.000, E1   -56.377, E3 +24282.641}
ENDSPLINE

SPLINE
SPL {X  -134.727, Y  +760.706, Z    +0.000, E1   -50.460, E3 +24470.873}
SPL {X  -155.580, Y  +711.748, Z    +0.000, E1   -32.084, E3 +24487.788}
SPL {X  -159.445, Y  +687.715, Z    +0.000, E1   -14.660, E3 +24490.634}
SPL {X  -159.995, Y  +675.725, Z    +0.000, E1    -3.424, E3 +24491.145}
SPL {X  -160.000, Y  +671.714, Z    +0.000, E1    +0.835, E3 +24491.186}
SPL {X  -160.000, Y  +663.084, Z    +0.000, E1   +21.134, E3 +24491.510}
SPL {X  -160.000, Y  +650.910, Z    +0.000, E1   +46.005, E3 +24492.664}
SPL {X  -160.000, Y  +634.843, Z    +0.000, E1   +61.273, E3 +24495.341}
SPL {X  -160.000, Y  +578.679, Z    +0.000, E1   +71.665, E3 +24513.174}
SPL {X  -160.000, Y  +387.528, Z    +0.000, E1   +73.487, E3 +24605.987}
SPL {X  -159.218, Y  +369.903, Z    +0.000, E1   +73.425, E3 +24617.854}
SPL {X  -156.808, Y  +353.900, Z    +0.000, E1   +73.180, E3 +24630.458}
SPL {X  -154.539, Y  +344.254, Z    +0.000, E1   +72.827, E3 +24639.995}
ENDSPLINE

SPLINE
SPL {X  -157.258, Y  +356.206, Z    +0.000, E1   +70.434, E3 +24654.567}
ENDSPLINE

SPLINE
SPL {X  -150.342, Y  +330.952, Z    +0.000, E1   +71.154, E3 +24666.240}
SPL {X  -141.358, Y  +310.748, Z    +0.000, E1   +71.233, E3 +24678.945}
SPL {X  -134.330, Y  +298.778, Z    +0.000, E1   +70.323, E3 +24692.793}
SPL {X  -128.957, Y  +290.989, Z    +0.000, E1   +69.528, E3 +24702.158}
SPL {X  -124.846, Y  +285.632, Z    +0.000, E1   +68.906, E3 +24708.621}
SPL {X  -121.783, Y  +281.927, Z    +0.000, E1   +68.403, E3 +24713.053}
SPL {X   -79.219, Y  +246.688, Z    +0.000, E1   +55.887, E3 +24834.560}
ENDSPLINE

SPLINE
SPL {X  -125.038, Y  +285.873, Z    +0.000, E1   +53.023, E3 +25011.601}
SPL {X  -149.949, Y  +329.886, Z    +0.000, E1   +41.515, E3 +25033.166}
SPL {X  -157.246, Y  +356.141, Z    +0.000, E1   +27.282, E3 +25038.223}
SPL {X  -159.525, Y  +373.376, Z    +0.000, E1   +13.812, E3 +25039.880}
SPL {X  -160.000, Y  +387.264, Z    +0.000, E1    +0.544, E3 +25040.337}
SPL {X  -160.000, Y  +390.384, Z    +0.000, E1    -6.008, E3 +25040.375}
SPL {X  -160.000, Y  +395.752, Z    +0.000, E1   -19.038, E3 +25040.568}
SPL {X  -160.000, Y  +404.289, Z    +0.000, E1   -38.292, E3 +25041.237}
SPL {X  -160.000, Y  +418.681, Z    +0.000, E1   -56.949, E3 +25043.426}
SPL {X  -160.000, Y  +471.977, Z    +0.000, E1   -70.792, E3 +25059.946}
SPL {X  -159.977, Y  +677.138, Z    +0.000, E1   -73.665, E3 +25156.437}
SPL {X  -157.805, Y  +700.810, Z    +0.000, E1   -73.511, E3 +25173.267}
SPL {X  -152.242, Y  +723.618, Z    +0.000, E1   -72.940, E3 +25193.180}
SPL {X  -145.929, Y  +740.010, Z    +0.000, E1   -72.229, E3 +25209.651}
SPL {X  -139.114, Y  +753.439, Z    +0.000, E1   -71.436, E3 +25224.290}
SPL {X  -132.333, Y  +764.333, Z    +0.000, E1   -70.535, E3 +25236.914}
SPL {X  -125.486, Y  +773.664, Z    +0.000, E1   -69.598, E3 +25247.888}
SPL {X  -121.321, Y  +778.713, Z    +0.000, E1   -68.872, E3 +25253.898}
SPL {X   -77.337, Y  +814.468, Z    +0.000, E1   -56.377, E3 +25372.529}
ENDSPLINE

SPLINE
SPL {X  -134.727, Y  +760.706, Z    +0.000, E1   -50.460, E3 +25560.761}
SPL {X  -155.580, Y  +711.748, Z    +0.000, E1   -32.084, E3 +25577.676}
SPL {X  -159.445, Y  +687.715, Z    +0.000, E1   -14.660, E3 +25580.522}
SPL {X  -159.995, Y  +675.725, Z    +0.000, E1    -3.424, E3 +25581.033}
SPL {X  -160.000, Y  +671.714, Z    +0.000, E1    +0.835, E3 +25581.074}
SPL {X  -160.000, Y  +663.084, Z    +0.000, E1   +21.134, E3 +25581.398}
SPL {X  -160.000, Y  +650.910, Z    +0.000, E1   +46.005, E3 +25582.552}
SPL {X  -160.000, Y  +634.843, Z    +0.000, E1   +61.273, E3 +25585.229}
SPL {X  -160.000, Y  +578.679, Z    +0.000, E1   +71.665, E3 +25603.062}
SPL {X  -160.000, Y  +387.528, Z    +0.000, E1   +73.487, E3 +25695.875}
SPL {X  -159.218, Y  +369.903, Z    +0.000, E1   +73.425, E3 +25707.742}
SPL {X  -156.808, Y  +353.900, Z    +0.000, E1   +73.180, E3 +25720.346}
SPL {X  -154.539, Y  +344.254, Z    +0.000, E1   +72.827, E3 +25729.883}
ENDSPLINE

SPLINE
SPL {X  -157.258, Y  +356.206, Z    +0.000, E1   +70.434, E3 +25744.455}
ENDSPLINE

SPLINE
SPL {X  -150.342, Y  +330.952, Z    +0.000, E1   +71.154, E3 +25756.128}
SPL {X  -141.358, Y  +310.748, Z    +0.000, E1   +71.233, E3 +25768.834}
SPL {X  -134.330, Y  +298.778, Z    +0.000, E1   +70.323, E3 +25782.681}
SPL {X  -128.957, Y  +290.989, Z    +0.000, E1   +69.528, E3 +25792.046}
SPL {X  -124.846, Y  +285.632, Z    +0.000, E1   +68.906, E3 +25798.509}
SPL {X  -121.783, Y  +281.927, Z    +0.000, E1   +68.403, E3 +25802.941}
SPL {X   -79.219, Y  +246.688, Z    +0.000, E1   +55.887, E3 +25924.448}
ENDSPLINE

SPLINE
SPL {X  -125.038, Y  +285.873, Z    +0.000, E1   +53.023, E3 +26101.489}
SPL {X  -149.949, Y  +329.886, Z    +0.000, E1   +41.515, E3 +26123.054}
SPL {X  -157.246, Y  +356.141, Z    +0.000, E1   +27.282, E3 +26128.111}
SPL {X  -159.525, Y  +373.376, Z    +0.000, E1   +13.812, E3 +26129.768}
SPL {X  -160.000, Y  +387.264, Z    +0.000, E1    +0.544, E3 +26130.225}
SPL {X  -160.000, Y  +390.384, Z    +0.000, E1    -6.008, E3 +26130.263}
SPL {X  -160.000, Y  +395.752, Z    +0.000, E1   -19.038, E3 +26130.456}
SPL {X  -160.000, Y  +404.289, Z    +0.000, E1   -38.292, E3 +26131.125}
SPL {X  -160.000, Y  +418.681, Z    +0.000, E1   -56.949, E3 +26133.314}
SPL {X  -160.000, Y  +471.977, Z    +0.000, E1   -70.792, E3 +26149.834}
SPL {X  -159.977, Y  +677.138, Z    +0.000, E1   -73.665, E3 +26246.325}
SPL {X  -157.805, Y  +700.810, Z    +0.000, E1   -73.511, E3 +26263.155}
SPL {X  -152.242, Y  +723.618, Z    +0.000, E1   -72.940, E3 +26283.068}
SPL {X  -145.929, Y  +740.010, Z    +0.000, E1   -72.229, E3 +26299.539}
SPL {X  -139.114, Y  +753.439, Z    +0.000, E1   -71.436, E3 +26314.178}
SPL {X  -132.333, Y  +764.333, Z    +0.000, E1   -70.535, E3 +26326.802}
SPL {X  -125.486, Y  +773.664, Z    +0.000, E1   -69.598, E3 +26337.776}
SPL {X  -121.321, Y  +778.713, Z    +0.000, E1   -68.872, E3 +26343.786}
SPL {X   -77.337, Y  +814.468, Z    +0.000, E1   -56.377, E3 +26462.417}
ENDSPLINE

SPLINE
SPL {X  -134.727, Y  +760.706, Z    +0.000, E1   -50.460, E3 +26650.649}
SPL {X  -155.580, Y  +711.748, Z    +0.000, E1   -32.084, E3 +26667.564}
SPL {X  -159.445, Y  +687.715, Z    +0.000, E1   -14.660, E3 +26670.411}
SPL {X  -159.995, Y  +675.725, Z    +0.000, E1    -3.424, E3 +26670.921}
SPL {X  -160.000, Y  +671.714, Z    +0.000, E1    +0.835, E3 +26670.962}
SPL {X  -160.000, Y  +663.084, Z    +0.000, E1   +21.134, E3 +26671.286}
SPL {X  -160.000, Y  +650.910, Z    +0.000, E1   +46.005, E3 +26672.440}
SPL {X  -160.000, Y  +634.843, Z    +0.000, E1   +61.273, E3 +26675.117}
SPL {X  -160.000, Y  +578.679, Z    +0.000, E1   +71.665, E3 +26692.950}
SPL {X  -160.000, Y  +387.528, Z    +0.000, E1   +73.487, E3 +26785.763}
SPL {X  -159.218, Y  +369.903, Z    +0.000, E1   +73.425, E3 +26797.630}
SPL {X  -156.808, Y  +353.900, Z    +0.000, E1   +73.180, E3 +26810.234}
SPL {X  -154.539, Y  +344.254, Z    +0.000, E1   +72.827, E3 +26819.771}
ENDSPLINE

SPLINE
SPL {X  -157.258, Y  +356.206, Z    +0.000, E1   +70.434, E3 +26834.344}
ENDSPLINE

SPLINE
SPL {X  -150.342, Y  +330.952, Z    +0.000, E1   +71.154, E3 +26846.016}
SPL {X  -141.358, Y  +310.748, Z    +0.000, E1   +71.233, E3 +26858.722}
SPL {X  -134.330, Y  +298.778, Z    +0.000, E1   +70.323, E3 +26872.569}
SPL {X  -128.957, Y  +290.989, Z    +0.000, E1   +69.528, E3 +26881.934}
SPL {X  -124.846, Y  +285.632, Z    +0.000, E1   +68.906, E3 +26888.397}
SPL {X  -121.783, Y  +281.927, Z    +0.000, E1   +68.403, E3 +26892.830}
SPL {X   -79.219, Y  +246.688, Z    +0.000, E1   +55.887, E3 +27014.336}
ENDSPLINE

SPLINE
SPL {X  -125.038, Y  +285.873, Z    +0.000, E1   +53.023, E3 +27191.377}
SPL {X  -149.949, Y  +329.886, Z    +0.000, E1   +41.515, E3 +27212.942}
SPL {X  -157.246, Y  +356.141, Z    +0.000, E1   +27.282, E3 +27217.999}
SPL {X  -159.525, Y  +373.376, Z    +0.000, E1   +13.812, E3 +27219.656}
SPL {X  -160.000, Y  +387.264, Z    +0.000, E1    +0.544, E3 +27220.113}
SPL {X  -160.000, Y  +390.384, Z    +0.000, E1    -6.008, E3 +27220.151}
SPL {X  -160.000, Y  +395.752, Z    +0.000, E1   -19.038, E3 +27220.344}
SPL {X  -160.000, Y  +404.289, Z    +0.000, E1   -38.292, E3 +27221.013}
SPL {X  -160.000, Y  +418.681, Z    +0.000, E1   -56.949, E3 +27223.202}
SPL {X  -160.000, Y  +471.977, Z    +0.000, E1   -70.792, E3 +27239.722}
SPL {X  -159.977, Y  +677.138, Z    +0.000, E1   -73.665, E3 +27336.213}
SPL {X  -157.805, Y  +700.810, Z    +0.000, E1   -73.511, E3 +27353.043}
SPL {X  -152.242, Y  +723.618, Z    +0.000, E1   -72.940, E3 +27372.956}
SPL {X  -145.929, Y  +740.010, Z    +0.000, E1   -72.229, E3 +27389.427}
SPL {X  -139.114, Y  +753.439, Z    +0.000, E1   -71.436, E3 +27404.066}
SPL {X  -132.333, Y  +764.333, Z    +0.000, E1   -70.535, E3 +27416.690}
SPL {X  -125.486, Y  +773.664, Z    +0.000, E1   -69.598, E3 +27427.664}
SPL {X  -121.321, Y  +778.713, Z    +0.000, E1   -68.872, E3 +27433.674}
SPL {X   -77.337, Y  +814.468, Z    +0.000, E1   -56.377, E3 +27552.305}
ENDSPLINE

SPLINE
SPL {X  -134.727, Y  +760.706, Z    +0.000, E1   -50.460, E3 +27740.537}
SPL {X  -155.580, Y  +711.748, Z    +0.000, E1   -32.084, E3 +27757.452}
SPL {X  -159.445, Y  +687.715, Z    +0.000, E1   -14.660, E3 +27760.299}
SPL {X  -159.995, Y  +675.725, Z    +0.000, E1    -3.424, E3 +27760.809}
SPL {X  -160.000, Y  +671.714, Z    +0.000, E1    +0.835, E3 +27760.850}
SPL {X  -160.000, Y  +663.084, Z    +0.000, E1   +21.134, E3 +27761.174}
SPL {X  -160.000, Y  +650.910, Z    +0.000, E1   +46.005, E3 +27762.328}
SPL {X  -160.000, Y  +634.843, Z    +0.000, E1   +61.273, E3 +27765.005}
SPL {X  -160.000, Y  +578.679, Z    +0.000, E1   +71.665, E3 +27782.838}
SPL {X  -160.000, Y  +387.528, Z    +0.000, E1   +73.487, E3 +27875.651}
SPL {X  -159.218, Y  +369.903, Z    +0.000, E1   +73.425, E3 +27887.518}
SPL {X  -156.808, Y  +353.900, Z    +0.000, E1   +73.180, E3 +27900.122}
SPL {X  -154.539, Y  +344.254, Z    +0.000, E1   +72.827, E3 +27909.659}
ENDSPLINE

SPLINE
SPL {X  -157.258, Y  +356.206, Z    +0.000, E1   +70.434, E3 +27924.232}
ENDSPLINE

SPLINE
SPL {X  -150.342, Y  +330.952, Z    +0.000, E1   +71.154, E3 +27935.904}
SPL {X  -141.358, Y  +310.748, Z    +0.000, E1   +71.233, E3 +27948.610}
SPL {X  -134.330, Y  +298.778, Z    +0.000, E1   +70.323, E3 +27962.457}
SPL {X  -128.957, Y  +290.989, Z    +0.000, E1   +69.528, E3 +27971.822}
SPL {X  -124.846, Y  +285.632, Z    +0.000, E1   +68.906, E3 +27978.285}
SPL {X  -121.783, Y  +281.927, Z    +0.000, E1   +68.403, E3 +27982.718}
SPL {X   -79.219, Y  +246.688, Z    +0.000, E1   +55.887, E3 +28104.224}
ENDSPLINE

SPLINE
SPL {X  -125.038, Y  +285.873, Z    +0.000, E1   +53.023, E3 +28281.265}
SPL {X  -149.949, Y  +329.886, Z    +0.000, E1   +41.515, E3 +28302.830}
SPL {X  -157.246, Y  +356.141, Z    +0.000, E1   +27.282, E3 +28307.887}
SPL {X  -159.525, Y  +373.376, Z    +0.000, E1   +13.812, E3 +28309.544}
SPL {X  -160.000, Y  +387.264, Z    +0.000, E1    +0.544, E3 +28310.002}
SPL {X  -160.000, Y  +390.384, Z    +0.000, E1    -6.008, E3 +28310.039}
SPL {X  -160.000, Y  +395.752, Z    +0.000, E1   -19.038, E3 +28310.232}
SPL {X  -160.000, Y  +404.289, Z    +0.000, E1   -38.292, E3 +28310.901}
SPL {X  -160.000, Y  +418.681, Z    +0.000, E1   -56.949, E3 +28313.090}
SPL {X  -160.000, Y  +471.977, Z    +0.000, E1   -70.792, E3 +28329.610}
SPL {X  -159.977, Y  +677.138, Z    +0.000, E1   -73.665, E3 +28426.101}
SPL {X  -157.805, Y  +700.810, Z    +0.000, E1   -73.511, E3 +28442.931}
SPL {X  -152.242, Y  +723.618, Z    +0.000, E1   -72.940, E3 +28462.844}
SPL {X  -145.929, Y  +740.010, Z    +0.000, E1   -72.229, E3 +28479.315}
SPL {X  -139.114, Y  +753.439, Z    +0.000, E1   -71.436, E3 +28493.954}
SPL {X  -132.333, Y  +764.333, Z    +0.000, E1   -70.535, E3 +28506.578}
SPL {X  -125.486, Y  +773.664, Z    +0.000, E1   -69.598, E3 +28517.552}
SPL {X  -121.321, Y  +778.713, Z    +0.000, E1   -68.872, E3 +28523.562}
SPL {X   -77.337, Y  +814.468, Z    +0.000, E1   -56.377, E3 +28642.193}
ENDSPLINE

SPLINE
SPL {X  -134.727, Y  +760.706, Z    +0.000, E1   -50.460, E3 +28830.425}
SPL {X  -155.580, Y  +711.748, Z    +0.000, E1   -32.084, E3 +28847.340}
SPL {X  -159.445, Y  +687.715, Z    +0.000, E1   -14.660, E3 +28850.187}
SPL {X  -159.995, Y  +675.725, Z    +0.000, E1    -3.424, E3 +28850.697}
SPL {X  -160.000, Y  +671.714, Z    +0.000, E1    +0.835, E3 +28850.738}
SPL {X  -160.000, Y  +663.084, Z    +0.000, E1   +21.134, E3 +28851.062}
SPL {X  -160.000, Y  +650.910, Z    +0.000, E1   +46.005, E3 +28852.216}
SPL {X  -160.000, Y  +634.843, Z    +0.000, E1   +61.273, E3 +28854.893}
SPL {X  -160.000, Y  +578.679, Z    +0.000, E1   +71.665, E3 +28872.726}
SPL {X  -160.000, Y  +387.528, Z    +0.000, E1   +73.487, E3 +28965.539}
SPL {X  -159.218, Y  +369.903, Z    +0.000, E1   +73.425, E3 +28977.406}
SPL {X  -156.808, Y  +353.900, Z    +0.000, E1   +73.180, E3 +28990.010}
SPL {X  -154.539, Y  +344.254, Z    +0.000, E1   +72.827, E3 +28999.547}
ENDSPLINE

SPLINE
SPL {X  -157.258, Y  +356.206, Z    +0.000, E1   +70.434, E3 +29014.120}
ENDSPLINE

SPLINE
SPL {X  -150.342, Y  +330.952, Z    +0.000, E1   +71.154, E3 +29025.792}
SPL {X  -141.358, Y  +310.748, Z    +0.000, E1   +71.233, E3 +29038.498}
SPL {X  -134.330, Y  +298.778, Z    +0.000, E1   +70.323, E3 +29052.345}
SPL {X  -128.957, Y  +290.989, Z    +0.000, E1   +69.528, E3 +29061.710}
SPL {X  -124.846, Y  +285.632, Z    +0.000, E1   +68.906, E3 +29068.173}
SPL {X  -121.783, Y  +281.927, Z    +0.000, E1   +68.403, E3 +29072.606}
SPL {X   -79.219, Y  +246.688, Z    +0.000, E1   +55.887, E3 +29194.112}
ENDSPLINE

SPLINE
SPL {X  -125.038, Y  +285.873, Z    +0.000, E1   +53.023, E3 +29371.153}
SPL {X  -149.949, Y  +329.886, Z    +0.000, E1   +41.515, E3 +29392.718}
SPL {X  -157.246, Y  +356.141, Z    +0.000, E1   +27.282, E3 +29397.775}
SPL {X  -159.525, Y  +373.376, Z    +0.000, E1   +13.812, E3 +29399.432}
SPL {X  -160.000, Y  +387.264, Z    +0.000, E1    +0.544, E3 +29399.890}
SPL {X  -160.000, Y  +390.384, Z    +0.000, E1    -6.008, E3 +29399.927}
SPL {X  -160.000, Y  +395.752, Z    +0.000, E1   -19.038, E3 +29400.120}
SPL {X  -160.000, Y  +404.289, Z    +0.000, E1   -38.292, E3 +29400.789}
SPL {X  -160.000, Y  +418.681, Z    +0.000, E1   -56.949, E3 +29402.979}
SPL {X  -160.000, Y  +471.977, Z    +0.000, E1   -70.792, E3 +29419.498}
SPL {X  -159.977, Y  +677.138, Z    +0.000, E1   -73.665, E3 +29515.989}
SPL {X  -157.805, Y  +700.810, Z    +0.000, E1   -73.511, E3 +29532.819}
SPL {X  -152.242, Y  +723.618, Z    +0.000, E1   -72.940, E3 +29552.732}
SPL {X  -145.929, Y  +740.010, Z    +0.000, E1   -72.229, E3 +29569.203}
SPL {X  -139.114, Y  +753.439, Z    +0.000, E1   -71.436, E3 +29583.842}
SPL {X  -132.333, Y  +764.333, Z    +0.000, E1   -70.535, E3 +29596.466}
SPL {X  -125.486, Y  +773.664, Z    +0.000, E1   -69.598, E3 +29607.440}
SPL {X  -121.321, Y  +778.713, Z    +0.000, E1   -68.872, E3 +29613.450}
SPL {X   -77.337, Y  +814.468, Z    +0.000, E1   -56.377, E3 +29732.081}
ENDSPLINE

SPLINE
SPL {X  -134.727, Y  +760.706, Z    +0.000, E1   -50.460, E3 +29920.313}
SPL {X  -155.580, Y  +711.748, Z    +0.000, E1   -32.084, E3 +29937.228}
SPL {X  -159.445, Y  +687.715, Z    +0.000, E1   -14.660, E3 +29940.075}
SPL {X  -159.995, Y  +675.725, Z    +0.000, E1    -3.424, E3 +29940.585}
SPL {X  -160.000, Y  +671.714, Z    +0.000, E1    +0.835, E3 +29940.626}
SPL {X  -160.000, Y  +663.084, Z    +0.000, E1   +21.134, E3 +29940.950}
SPL {X  -160.000, Y  +650.910, Z    +0.000, E1   +46.005, E3 +29942.104}
SPL {X  -160.000, Y  +634.843, Z    +0.000, E1   +61.273, E3 +29944.781}
SPL {X  -160.000, Y  +578.679, Z    +0.000, E1   +71.665, E3 +29962.614}
SPL {X  -160.000, Y  +387.528, Z    +0.000, E1   +73.487, E3 +30055.427}
SPL {X  -159.218, Y  +369.903, Z    +0.000, E1   +73.425, E3 +30067.294}
SPL {X  -156.808, Y  +353.900, Z    +0.000, E1   +73.180, E3 +30079.898}
SPL {X  -154.539, Y  +344.254, Z    +0.000, E1   +72.827, E3 +30089.435}
ENDSPLINE

SPLINE
SPL {X  -157.258, Y  +356.206, Z    +0.000, E1   +70.434, E3 +30104.008}
ENDSPLINE

SPLINE
SPL {X  -150.342, Y  +330.952, Z    +0.000, E1   +71.154, E3 +30115.680}
SPL {X  -141.358, Y  +310.748, Z    +0.000, E1   +71.233, E3 +30128.386}
SPL {X  -134.330, Y  +298.778, Z    +0.000, E1   +70.323, E3 +30142.233}
SPL {X  -128.957, Y  +290.989, Z    +0.000, E1   +69.528, E3 +30151.598}
SPL {X  -124.846, Y  +285.632, Z    +0.000, E1   +68.906, E3 +30158.061}
SPL {X  -121.783, Y  +281.927, Z    +0.000, E1   +68.403, E3 +30162.494}
SPL {X   -79.219, Y  +246.688, Z    +0.000, E1   +55.887, E3 +30284.000}
ENDSPLINE

SPLINE
SPL {X  -125.038, Y  +285.873, Z    +0.000, E1   +53.023, E3 +30461.041}
SPL {X  -149.949, Y  +329.886, Z    +0.000, E1   +41.515, E3 +30482.606}
SPL {X  -157.246, Y  +356.141, Z    +0.000, E1   +27.282, E3 +30487.663}
SPL {X  -159.525, Y  +373.376, Z    +0.000, E1   +13.812, E3 +30489.320}
SPL {X  -160.000, Y  +387.264, Z    +0.000, E1    +0.544, E3 +30489.778}
SPL {X  -160.000, Y  +390.384, Z    +0.000, E1    -6.008, E3 +30489.815}
SPL {X  -160.000, Y  +395.752, Z    +0.000, E1   -19.038, E3 +30490.008}
SPL {X  -160.000, Y  +404.289, Z    +0.000, E1   -38.292, E3 +30490.677}
SPL {X  -160.000, Y  +418.681, Z    +0.000, E1   -56.949, E3 +30492.867}
SPL {X  -160.000, Y  +471.977, Z    +0.000, E1   -70.792, E3 +30509.386}
SPL {X  -159.977, Y  +677.138, Z    +0.000, E1   -73.665, E3 +30605.877}
SPL {X  -157.805, Y  +700.810, Z    +0.000, E1   -73.511, E3 +30622.707}
SPL {X  -152.242, Y  +723.618, Z    +0.000, E1   -72.940, E3 +30642.620}
SPL {X  -145.929, Y  +740.010, Z    +0.000, E1   -72.229, E3 +30659.091}
SPL {X  -139.114, Y  +753.439, Z    +0.000, E1   -71.436, E3 +30673.730}
SPL {X  -132.333, Y  +764.333, Z    +0.000, E1   -70.535, E3 +30686.354}
SPL {X  -125.486, Y  +773.664, Z    +0.000, E1   -69.598, E3 +30697.328}
SPL {X  -121.321, Y  +778.713, Z    +0.000, E1   -68.872, E3 +30703.338}
SPL {X   -77.337, Y  +814.468, Z    +0.000, E1   -56.377, E3 +30821.969}
ENDSPLINE

SPLINE
SPL {X  -134.727, Y  +760.706, Z    +0.000, E1   -50.460, E3 +31010.201}
SPL {X  -155.580, Y  +711.748, Z    +0.000, E1   -32.084, E3 +31027.116}
SPL {X  -159.445, Y  +687.715, Z    +0.000, E1   -14.660, E3 +31029.963}
SPL {X  -159.995, Y  +675.725, Z    +0.000, E1    -3.424, E3 +31030.473}
SPL {X  -160.000, Y  +671.714, Z    +0.000, E1    +0.835, E3 +31030.514}
SPL {X  -160.000, Y  +663.084, Z    +0.000, E1   +21.134, E3 +31030.838}
SPL {X  -160.000, Y  +650.910, Z    +0.000, E1   +46.005, E3 +31031.992}
SPL {X  -160.000, Y  +634.843, Z    +0.000, E1   +61.273, E3 +31034.669}
SPL {X  -160.000, Y  +578.679, Z    +0.000, E1   +71.665, E3 +31052.502}
SPL {X  -160.000, Y  +387.528, Z    +0.000, E1   +73.487, E3 +31145.315}
SPL {X  -159.218, Y  +369.903, Z    +0.000, E1   +73.425, E3 +31157.182}
SPL {X  -156.808, Y  +353.900, Z    +0.000, E1   +73.180, E3 +31169.786}
SPL {X  -154.539, Y  +344.254, Z    +0.000, E1   +72.827, E3 +31179.323}
ENDSPLINE

SPLINE
SPL {X  -157.258, Y  +356.206, Z    +0.000, E1   +70.434, E3 +31193.896}
ENDSPLINE

SPLINE
SPL {X  -150.342, Y  +330.952, Z    +0.000, E1   +71.154, E3 +31205.568}
SPL {X  -141.358, Y  +310.748, Z    +0.000, E1   +71.233, E3 +31218.274}
SPL {X  -134.330, Y  +298.778, Z    +0.000, E1   +70.323, E3 +31232.121}
SPL {X  -128.957, Y  +290.989, Z    +0.000, E1   +69.528, E3 +31241.486}
SPL {X  -124.846, Y  +285.632, Z    +0.000, E1   +68.906, E3 +31247.949}
SPL {X  -121.783, Y  +281.927, Z    +0.000, E1   +68.403, E3 +31252.382}
SPL {X   -79.219, Y  +246.688, Z    +0.000, E1   +55.887, E3 +31373.888}
ENDSPLINE

SPLINE
SPL {X  -125.038, Y  +285.873, Z    +0.000, E1   +53.023, E3 +31550.929}
SPL {X  -149.949, Y  +329.886, Z    +0.000, E1   +41.515, E3 +31572.494}
SPL {X  -157.246, Y  +356.141, Z    +0.000, E1   +27.282, E3 +31577.551}
SPL {X  -159.525, Y  +373.376, Z    +0.000, E1   +13.812, E3 +31579.208}
SPL {X  -160.000, Y  +387.264, Z    +0.000, E1    +0.544, E3 +31579.666}
SPL {X  -160.000, Y  +390.384, Z    +0.000, E1    -6.008, E3 +31579.703}
SPL {X  -160.000, Y  +395.752, Z    +0.000, E1   -19.038, E3 +31579.896}
SPL {X  -160.000, Y  +404.289, Z    +0.000, E1   -38.292, E3 +31580.565}
SPL {X  -160.000, Y  +418.681, Z    +0.000, E1   -56.949, E3 +31582.755}
SPL {X  -160.000, Y  +471.977, Z    +0.000, E1   -70.792, E3 +31599.274}
SPL {X  -159.977, Y  +677.138, Z    +0.000, E1   -73.665, E3 +31695.765}
SPL {X  -157.805, Y  +700.810, Z    +0.000, E1   -73.511, E3 +31712.595}
SPL {X  -152.242, Y  +723.618, Z    +0.000, E1   -72.940, E3 +31732.508}
SPL {X  -145.929, Y  +740.010, Z    +0.000, E1   -72.229, E3 +31748.979}
SPL {X  -139.114, Y  +753.439, Z    +0.000, E1   -71.436, E3 +31763.618}
SPL {X  -132.333, Y  +764.333, Z    +0.000, E1   -70.535, E3 +31776.242}
SPL {X  -125.486, Y  +773.664, Z    +0.000, E1   -69.598, E3 +31787.216}
SPL {X  -121.321, Y  +778.713, Z    +0.000, E1   -68.872, E3 +31793.226}
SPL {X   -77.337, Y  +814.468, Z    +0.000, E1   -56.377, E3 +31911.857}
ENDSPLINE

SPLINE
SPL {X  -134.727, Y  +760.706, Z    +0.000, E1   -50.460, E3 +32100.089}
SPL {X  -155.580, Y  +711.748, Z    +0.000, E1   -32.084, E3 +32117.004}
SPL {X  -159.445, Y  +687.715, Z    +0.000, E1   -14.660, E3 +32119.851}
SPL {X  -159.995, Y  +675.725, Z    +0.000, E1    -3.424, E3 +32120.361}
SPL {X  -160.000, Y  +671.714, Z    +0.000, E1    +0.835, E3 +32120.402}
SPL {X  -160.000, Y  +663.084, Z    +0.000, E1   +21.134, E3 +32120.726}
SPL {X  -160.000, Y  +650.910, Z    +0.000, E1   +46.005, E3 +32121.880}
SPL {X  -160.000, Y  +634.843, Z    +0.000, E1   +61.273, E3 +32124.557}
SPL {X  -160.000, Y  +578.679, Z    +0.000, E1   +71.665, E3 +32142.391}
SPL {X  -160.000, Y  +387.528, Z    +0.000, E1   +73.487, E3 +32235.203}
SPL {X  -159.218, Y  +369.903, Z    +0.000, E1   +73.425, E3 +32247.070}
SPL {X  -156.808, Y  +353.900, Z    +0.000, E1   +73.180, E3 +32259.674}
SPL {X  -154.539, Y  +344.254, Z    +0.000, E1   +72.827, E3 +32269.211}
ENDSPLINE

SPLINE
SPL {X  -157.258, Y  +356.206, Z    +0.000, E1   +70.434, E3 +32283.784}
ENDSPLINE

SPLINE
SPL {X  -150.342, Y  +330.952, Z    +0.000, E1   +71.154, E3 +32295.456}
SPL {X  -141.358, Y  +310.748, Z    +0.000, E1   +71.233, E3 +32308.162}
SPL {X  -134.330, Y  +298.778, Z    +0.000, E1   +70.323, E3 +32322.009}
SPL {X  -128.957, Y  +290.989, Z    +0.000, E1   +69.528, E3 +32331.374}
SPL {X  -124.846, Y  +285.632, Z    +0.000, E1   +68.906, E3 +32337.837}
SPL {X  -121.783, Y  +281.927, Z    +0.000, E1   +68.403, E3 +32342.270}
SPL {X   -79.219, Y  +246.688, Z    +0.000, E1   +55.887, E3 +32463.776}
ENDSPLINE

SPLINE
SPL {X  -125.038, Y  +285.873, Z    +0.000, E1   +53.023, E3 +32640.817}
SPL {X  -149.949, Y  +329.886, Z    +0.000, E1   +41.515, E3 +32662.382}
SPL {X  -157.246, Y  +356.141, Z    +0.000, E1   +27.282, E3 +32667.439}
SPL {X  -159.525, Y  +373.376, Z    +0.000, E1   +13.812, E3 +32669.096}
SPL {X  -160.000, Y  +387.264, Z    +0.000, E1    +0.544, E3 +32669.554}
SPL {X  -160.000, Y  +390.384, Z    +0.000, E1    -6.008, E3 +32669.591}
SPL {X  -160.000, Y  +395.752, Z    +0.000, E1   -19.038, E3 +32669.784}
SPL {X  -160.000, Y  +404.289, Z    +0.000, E1   -38.292, E3 +32670.453}
SPL {X  -160.000, Y  +418.681, Z    +0.000, E1   -56.949, E3 +32672.643}
SPL {X  -160.000, Y  +458.961, Z    +0.000, E1   -69.778, E3 +32684.239}
SPL {X  -160.000, Y  +485.343, Z    +0.000, E1   -71.539, E3 +32694.225}
SPL {X  -159.977, Y  +677.138, Z    +0.000, E1   -73.665, E3 +32785.653}
SPL {X  -157.805, Y  +700.810, Z    +0.000, E1   -73.511, E3 +32802.483}
SPL {X  -152.242, Y  +723.618, Z    +0.000, E1   -72.940, E3 +32822.396}
SPL {X  -145.929, Y  +740.010, Z    +0.000, E1   -72.229, E3 +32838.867}
SPL {X  -139.114, Y  +753.439, Z    +0.000, E1   -71.436, E3 +32853.506}
SPL {X  -132.333, Y  +764.333, Z    +0.000, E1   -70.535, E3 +32866.130}
SPL {X  -125.486, Y  +773.664, Z    +0.000, E1   -69.598, E3 +32877.104}
SPL {X  -121.321, Y  +778.713, Z    +0.000, E1   -68.872, E3 +32883.114}
SPL {X   -77.337, Y  +814.468, Z    +0.000, E1   -56.377, E3 +33001.745}
ENDSPLINE

SPLINE
SPL {X  -134.727, Y  +760.706, Z    +0.000, E1   -50.460, E3 +33189.977}
SPL {X  -155.580, Y  +711.748, Z    +0.000, E1   -32.084, E3 +33206.892}
SPL {X  -159.445, Y  +687.715, Z    +0.000, E1   -14.660, E3 +33209.739}
SPL {X  -159.995, Y  +675.725, Z    +0.000, E1    -3.424, E3 +33210.250}
SPL {X  -160.000, Y  +671.714, Z    +0.000, E1    +0.835, E3 +33210.290}
SPL {X  -160.000, Y  +663.084, Z    +0.000, E1   +21.134, E3 +33210.614}
SPL {X  -160.000, Y  +650.910, Z    +0.000, E1   +46.005, E3 +33211.768}
SPL {X  -160.000, Y  +634.843, Z    +0.000, E1   +61.273, E3 +33214.445}
SPL {X  -160.000, Y  +578.679, Z    +0.000, E1   +71.665, E3 +33232.279}
SPL {X  -160.000, Y  +387.528, Z    +0.000, E1   +73.487, E3 +33325.091}
SPL {X  -159.218, Y  +369.903, Z    +0.000, E1   +73.425, E3 +33336.958}
SPL {X  -156.808, Y  +353.900, Z    +0.000, E1   +73.180, E3 +33349.562}
SPL {X  -154.539, Y  +344.254, Z    +0.000, E1   +72.827, E3 +33359.099}
ENDSPLINE

SPLINE
SPL {X  -157.258, Y  +356.206, Z    +0.000, E1   +70.434, E3 +33373.672}
ENDSPLINE

SPLINE
SPL {X  -150.342, Y  +330.952, Z    +0.000, E1   +71.154, E3 +33385.344}
SPL {X  -141.358, Y  +310.748, Z    +0.000, E1   +71.233, E3 +33398.050}
SPL {X  -134.330, Y  +298.778, Z    +0.000, E1   +70.323, E3 +33411.897}
SPL {X  -128.957, Y  +290.989, Z    +0.000, E1   +69.528, E3 +33421.262}
SPL {X  -124.846, Y  +285.632, Z    +0.000, E1   +68.906, E3 +33427.726}
SPL {X  -121.783, Y  +281.927, Z    +0.000, E1   +68.403, E3 +33432.158}
SPL {X   -79.219, Y  +246.688, Z    +0.000, E1   +55.887, E3 +33553.664}
ENDSPLINE

SPLINE
SPL {X  -125.038, Y  +285.873, Z    +0.000, E1   +53.023, E3 +33730.705}
SPL {X  -149.949, Y  +329.886, Z    +0.000, E1   +41.515, E3 +33752.270}
SPL {X  -157.246, Y  +356.141, Z    +0.000, E1   +27.282, E3 +33757.327}
SPL {X  -159.525, Y  +373.376, Z    +0.000, E1   +13.812, E3 +33758.984}
SPL {X  -160.000, Y  +387.264, Z    +0.000, E1    +0.544, E3 +33759.442}
SPL {X  -160.000, Y  +390.384, Z    +0.000, E1    -6.008, E3 +33759.479}
SPL {X  -160.000, Y  +395.752, Z    +0.000, E1   -19.038, E3 +33759.673}
SPL {X  -160.000, Y  +404.289, Z    +0.000, E1   -38.292, E3 +33760.341}
SPL {X  -160.000, Y  +418.681, Z    +0.000, E1   -56.949, E3 +33762.531}
SPL {X  -160.000, Y  +471.977, Z    +0.000, E1   -70.792, E3 +33779.050}
SPL {X  -159.977, Y  +677.138, Z    +0.000, E1   -73.665, E3 +33875.541}
SPL {X  -157.805, Y  +700.810, Z    +0.000, E1   -73.511, E3 +33892.371}
SPL {X  -152.242, Y  +723.618, Z    +0.000, E1   -72.940, E3 +33912.284}
SPL {X  -145.929, Y  +740.010, Z    +0.000, E1   -72.229, E3 +33928.756}
SPL {X  -139.114, Y  +753.439, Z    +0.000, E1   -71.436, E3 +33943.394}
SPL {X  -132.333, Y  +764.333, Z    +0.000, E1   -70.535, E3 +33956.018}
SPL {X  -125.486, Y  +773.664, Z    +0.000, E1   -69.598, E3 +33966.992}
SPL {X  -121.321, Y  +778.713, Z    +0.000, E1   -68.872, E3 +33973.002}
SPL {X   -77.337, Y  +814.468, Z    +0.000, E1   -56.377, E3 +34091.633}
ENDSPLINE

SPLINE
SPL {X  -134.727, Y  +760.706, Z    +0.000, E1   -50.460, E3 +34279.865}
SPL {X  -155.580, Y  +711.748, Z    +0.000, E1   -32.084, E3 +34296.780}
SPL {X  -159.445, Y  +687.715, Z    +0.000, E1   -14.660, E3 +34299.627}
SPL {X  -159.995, Y  +675.725, Z    +0.000, E1    -3.424, E3 +34300.138}
SPL {X  -160.000, Y  +671.714, Z    +0.000, E1    +0.835, E3 +34300.178}
SPL {X  -160.000, Y  +663.084, Z    +0.000, E1   +21.134, E3 +34300.502}
SPL {X  -160.000, Y  +650.910, Z    +0.000, E1   +46.005, E3 +34301.656}
SPL {X  -160.000, Y  +634.843, Z    +0.000, E1   +61.273, E3 +34304.333}
SPL {X  -160.000, Y  +578.679, Z    +0.000, E1   +71.665, E3 +34322.167}
SPL {X  -160.000, Y  +387.528, Z    +0.000, E1   +73.487, E3 +34414.979}
SPL {X  -159.218, Y  +369.903, Z    +0.000, E1   +73.425, E3 +34426.846}
SPL {X  -156.808, Y  +353.900, Z    +0.000, E1   +73.180, E3 +34439.450}
SPL {X  -154.539, Y  +344.254, Z    +0.000, E1   +72.827, E3 +34448.987}
ENDSPLINE

SPLINE
SPL {X  -157.258, Y  +356.206, Z    +0.000, E1   +70.434, E3 +34463.560}
ENDSPLINE

SPLINE
SPL {X  -150.342, Y  +330.952, Z    +0.000, E1   +71.154, E3 +34475.232}
SPL {X  -141.358, Y  +310.748, Z    +0.000, E1   +71.233, E3 +34487.938}
SPL {X  -134.330, Y  +298.778, Z    +0.000, E1   +70.323, E3 +34501.785}
SPL {X  -128.957, Y  +290.989, Z    +0.000, E1   +69.528, E3 +34511.150}
SPL {X  -124.846, Y  +285.632, Z    +0.000, E1   +68.906, E3 +34517.614}
SPL {X  -121.783, Y  +281.927, Z    +0.000, E1   +68.403, E3 +34522.046}
SPL {X   -79.219, Y  +246.688, Z    +0.000, E1   +55.887, E3 +34643.552}
ENDSPLINE

SPLINE
SPL {X  -125.038, Y  +285.873, Z    +0.000, E1   +53.023, E3 +34820.593}
SPL {X  -149.949, Y  +329.886, Z    +0.000, E1   +41.515, E3 +34842.158}
SPL {X  -157.246, Y  +356.141, Z    +0.000, E1   +27.282, E3 +34847.215}
SPL {X  -159.525, Y  +373.376, Z    +0.000, E1   +13.812, E3 +34848.872}
SPL {X  -160.000, Y  +387.264, Z    +0.000, E1    +0.544, E3 +34849.330}
SPL {X  -160.000, Y  +390.384, Z    +0.000, E1    -6.008, E3 +34849.367}
SPL {X  -160.000, Y  +395.752, Z    +0.000, E1   -19.038, E3 +34849.561}
SPL {X  -160.000, Y  +404.289, Z    +0.000, E1   -38.292, E3 +34850.229}
SPL {X  -160.000, Y  +418.681, Z    +0.000, E1   -56.949, E3 +34852.419}
SPL {X  -160.000, Y  +471.977, Z    +0.000, E1   -70.792, E3 +34868.938}
SPL {X  -159.977, Y  +677.138, Z    +0.000, E1   -73.665, E3 +34965.429}
SPL {X  -157.805, Y  +700.810, Z    +0.000, E1   -73.511, E3 +34982.259}
SPL {X  -152.242, Y  +723.618, Z    +0.000, E1   -72.940, E3 +35002.172}
SPL {X  -145.929, Y  +740.010, Z    +0.000, E1   -72.229, E3 +35018.644}
SPL {X  -139.114, Y  +753.439, Z    +0.000, E1   -71.436, E3 +35033.282}
SPL {X  -132.333, Y  +764.333, Z    +0.000, E1   -70.535, E3 +35045.906}
SPL {X  -125.486, Y  +773.664, Z    +0.000, E1   -69.598, E3 +35056.880}
SPL {X  -121.321, Y  +778.713, Z    +0.000, E1   -68.872, E3 +35062.890}
SPL {X   -77.337, Y  +814.468, Z    +0.000, E1   -56.377, E3 +35181.521}
ENDSPLINE

SPLINE
SPL {X  -134.727, Y  +760.706, Z    +0.000, E1   -50.460, E3 +35369.753}
SPL {X  -155.580, Y  +711.748, Z    +0.000, E1   -32.084, E3 +35386.668}
SPL {X  -159.445, Y  +687.715, Z    +0.000, E1   -14.660, E3 +35389.515}
SPL {X  -159.995, Y  +675.725, Z    +0.000, E1    -3.424, E3 +35390.026}
SPL {X  -160.000, Y  +671.714, Z    +0.000, E1    +0.835, E3 +35390.066}
SPL {X  -160.000, Y  +663.084, Z    +0.000, E1   +21.134, E3 +35390.390}
SPL {X  -160.000, Y  +650.910, Z    +0.000, E1   +46.005, E3 +35391.544}
SPL {X  -160.000, Y  +634.843, Z    +0.000, E1   +61.273, E3 +35394.221}
SPL {X  -160.000, Y  +578.679, Z    +0.000, E1   +71.665, E3 +35412.055}
SPL {X  -160.000, Y  +387.528, Z    +0.000, E1   +73.487, E3 +35504.867}
SPL {X  -159.218, Y  +369.903, Z    +0.000, E1   +73.425, E3 +35516.734}
SPL {X  -156.808, Y  +353.900, Z    +0.000, E1   +73.180, E3 +35529.338}
SPL {X  -154.539, Y  +344.254, Z    +0.000, E1   +72.827, E3 +35538.875}
ENDSPLINE

SPLINE
SPL {X  -157.258, Y  +356.206, Z    +0.000, E1   +70.434, E3 +35553.448}
ENDSPLINE

